# B&R Automation Studio project vibratorControlWithCurrentController (part 6)

#### Main.st - Init, cyclic, exit code
```iecst
PROGRAM _INIT

	cm.setup.name := 'sampling';

END_PROGRAM

PROGRAM _CYCLIC

	interface ACCESS ADR(gCapconInterface);

	IF gMainInterface.status.simulation OR gSimulation.status.simulateAllButWing THEN
		executeSim;
	END_IF

	IF interface.status.reset THEN
		interface.status.reset := FALSE;
		this.sim.state := 0;
	END_IF

	// ************************************************ //
	// *************** Wing Sampling ****************** //
	// ************************************************ //
	IF NOT this.hw.di_upperFlap_change THEN
		this.WingHwTOFs[0].OUT := FALSE;
	END_IF

	IF NOT this.hw.di_middleFlap_change THEN
		this.WingHwTOFs[1].OUT := FALSE;
	END_IF

	IF NOT this.hw.di_bottomFlap_change THEN
		this.WingHwTOFs[2].OUT := FALSE;
	END_IF

	IF NOT this.hw.di_neigbourFlap_change THEN
		this.WingHwTOFs[3].OUT := FALSE;
	END_IF

	FOR i:=0 TO 3 BY 1 DO
		IF NOT this.WingHwTOFs[i].OUT THEN
			this.WingHwTOFs[i].ET := this.WingHwTOFs[i].ET +1600; // 0.8 ms
		END_IF
		IF (this.WingHwTOFs[i].ET >= this.WingHwTOFs[i].PT) THEN
			CASE i OF

				0:
					IF this.hw.di_upperFlap_change THEN // only reset if changeOver signal is 1 again.
						this.WingHwTOFs[i].OUT := TRUE;
						this.WingHwTOFs[i].ET := 0;
					END_IF

				1:
					IF this.hw.di_middleFlap_change THEN // only reset if changeOver signal is 1 again.
						this.WingHwTOFs[i].OUT := TRUE;
						this.WingHwTOFs[i].ET := 0;
					END_IF

				2:
					IF this.hw.di_bottomFlap_change THEN // only reset if changeOver signal is 1 again.
						this.WingHwTOFs[i].OUT := TRUE;
						this.WingHwTOFs[i].ET := 0;
					END_IF

				3:
					IF this.hw.di_neigbourFlap_change THEN // only reset if changeOver signal is 1 again.
						this.WingHwTOFs[i].OUT := TRUE;
						this.WingHwTOFs[i].ET := 0;
					END_IF

			END_CASE
		END_IF
	END_FOR

	// ************************************************ //
	// ************** CAPCON ALGORITHM **************** //
	// ************************************************ //
	this.hw.ai_signal[0] := (this.hw.ai_signal[1]+this.lastAiSignal)/2;
	this.lastAiSignal := this.hw.ai_signal[1];
	FOR k:=0 TO 1 DO
		this.MTBasicsTimeDelay_capcon.Enable 	 := TRUE;
		this.MTBasicsTimeDelay_capcon.DelayTime  := 0.032;
		this.MTBasicsTimeDelay_capcon.In 		 := this.hw.ai_signal[k];
		this.MTBasicsTimeDelay_capcon();

		this.MTFilterMovingAverage_capcon.Enable		:= TRUE;
		this.MTFilterMovingAverage_capcon.WindowLength  := 40;
		this.MTFilterMovingAverage_capcon.In 			:= this.hw.ai_signal[k];
		this.MTFilterMovingAverage_capcon();

		this.BrickDetector_0.enable 	:= TRUE;
		this.BrickDetector_0.signal 	:= this.MTFilterMovingAverage_capcon.Out;
		this.BrickDetector_0.threshold 	:= gCapconInterface.status.capconMinThreshold;		 //15;
		this.BrickDetector_0.factorRmsMax := gCapconInterface.status.factorRmsMax;
		this.BrickDetector_0();

		this.CapconNoiseMeassure_0.beltSpeed := gBeltInterface.status.speed;
		this.CapconNoiseMeassure_0.rms := this.BrickDetector_0.rms;
		this.CapconNoiseMeassure_0();

		CASE cm.substate OF
			0:
				cm.description := 'wait for brick';

				this.BrickIntegral_0.enable := FALSE;
				this.BrickIntegral_0.calculate := FALSE;
				this.BrickIntegral_0();

				IF this.BrickDetector_0.brickCandidate AND NOT gMainInterface.status.emptying THEN
					this.BrickIntegral_0.baselineStart := this.BrickDetector_0.signal;
					cm.substate := 10;
				END_IF
			10:
				cm.description := 'measure brick';

				this.BrickIntegral_0.enable := TRUE;
				this.BrickIntegral_0.calculate := FALSE;
				this.BrickIntegral_0.signal := this.MTBasicsTimeDelay_capcon.Out;
				this.BrickIntegral_0();

				IF NOT this.BrickDetector_0.brickCandidate THEN
					cm.substate := 0;
				ELSIF this.BrickDetector_0.brickPresent THEN
					cm.substate := 20;
				END_IF

			20:
				cm.description := 'measure brick and wait for brick not present';

				this.BrickIntegral_0.enable := TRUE;
				this.BrickIntegral_0.calculate := FALSE;
				this.BrickIntegral_0.signal := this.MTBasicsTimeDelay_capcon.Out;
				this.BrickIntegral_0();

				IF this.BrickDetector_0.brickNotPresent THEN
					this.BrickIntegral_0.baselineEnd := this.BrickDetector_0.signal;
					this.BrickDetector_0.rmsMaxThreshold := this.BrickDetector_0.currentRmsMax;
					cm.substate := 30;
				END_IF

			30:
				cm.description := 'calculate integral';

				this.BrickIntegral_0.calculate := TRUE;
				this.BrickIntegral_0();

				IF this.BrickIntegral_0.done THEN
					this.BrickIntegral_0.calculate := FALSE;
					this.integralSum := this.integralSum + this.BrickIntegral_0.integral;

					cm.substate := 40;
				END_IF

			40:
				cm.description := 'Add peak integrals to array';

				IF this.BrickIntegral_0.noPeaks > 0 THEN
					FOR i:=0 TO this.BrickIntegral_0.noPeaks - 1 DO
						IF this.noPeaks <= MAX_PEAKS THEN
							this.peakIntegral[this.noPeaks] := this.BrickIntegral_0.integrals[i];
							this.noPeaks := this.noPeaks + 1;
						END_IF;
					END_FOR
				END_IF

				interface.status.noPeaks 	   := this.noPeaks;
				interface.status.peakIntegral  := this.peakIntegral;

				cm.substate := 50;

			50:
				cm.description := 'Verify peak integrals';

				this.VerifyPeaks_0.teachIntegral 	:= interface.status.teachIntegral;
				this.VerifyPeaks_0.controlPercent 	:= interface.parameter.controlPercent;
				this.VerifyPeaks_0.peakIntegral 	:= ADR(this.peakIntegral);
				this.VerifyPeaks_0.noPeaks			:= this.noPeaks;
				this.VerifyPeaks_0();

				interface.status.noVerifiedPeaks 	:= this.VerifyPeaks_0.noVerifiedPeaks;
				interface.status.verifiedPeakCount 	:= this.VerifyPeaks_0.peakCount;

				cm.substate := 60;

			60:
				cm.description := 'Verify adaptive peak integrals';

				this.VerifyPeaks_1.teachIntegral 	:= interface.status.adaptiveTeachIntegral;
				this.VerifyPeaks_1.controlPercent 	:= interface.parameter.controlPercent;
				this.VerifyPeaks_1.peakIntegral 	:= ADR(this.peakIntegral);
				this.VerifyPeaks_1.noPeaks			:= this.noPeaks;
				this.VerifyPeaks_1();

				interface.status.noAdaptiveVerifiedPeaks := this.VerifyPeaks_1.noVerifiedPeaks;

				cm.substate := 0;

		END_CASE
	END_FOR

	IF EDGEPOS(interface.status.ready) THEN
		this.integralSum := 0;
		this.brickError := FALSE;
		this.noPeaks := 0;
		this.noVerifiedPeaks := 0;
		interface.status.noPeaks := 0;
		interface.status.noVerifiedPeaks := 0;
		interface.status.noAdaptiveVerifiedPeaks := 0;
		FOR i:=0 TO MAX_PEAKS DO
			this.peakIntegral[i] := 0;
		END_FOR
	END_IF

	interface.status.integralSum := this.integralSum;
	interface.status.brickDetected := cm.substate >= 10;
	interface.status.brickPresent := cm.substate >= 20;

	// Test from FAT
	IF gCapconInterface.cmd.startSpeedSignalTest THEN
		IF NOT this.TON_0.IN THEN
			this.maxSignal := -30000;
			this.minSignal := 30000;
		END_IF

		// Save highest speed doing 5sec
		this.TON_0.PT := T#5s;
		this.TON_0.IN := TRUE;
		this.TON_0();
		this.maxSignal := SEL(this.hw.ai_signal[0]>this.maxSignal,this.maxSignal,this.hw.ai_signal[0]);
		this.minSignal := SEL(this.hw.ai_signal[0]<this.minSignal,this.minSignal,this.hw.ai_signal[0]);

		IF this.TON_0.Q THEN
			this.TON_0(IN:=FALSE);
			gCapconInterface.status.maxRawSignal := this.maxSignal-this.minSignal; // max signal peak-to-peak
			IF gCapconInterface.status.maxRawSignal > 5000 THEN
				gCapconInterface.status.maxRawSignal := 0;
			END_IF
			gCapconInterface.cmd.startSpeedSignalTest := FALSE;
		END_IF
	END_IF

END_PROGRAM

PROGRAM _EXIT

END_PROGRAM
```

#### executeSim.st
```iecst
ACTION executeSim:

	this.hw.ai_signal[1] := gSimCapcon.status.simSignal;

END_ACTION
```

#### Types.typ - Local data types
```iecst
TYPE
	local_alarm_typ : 	STRUCT
		noisePeakPeak : BOOL;
		noiseOffset : BOOL;
		noiseSpeed : BOOL;
	END_STRUCT;
	local_TOF_typ : 	STRUCT
		PT : UDINT := 10000; (*10ms*)
		ET : UDINT;
		OUT : BOOL;
	END_STRUCT;
	local_brickDetect_typ : 	STRUCT
		state : USINT;
		stateDescription : STRING[200];
	END_STRUCT;
	local_typ : 	STRUCT
		hw : local_hw_typ;
		sim : local_sim_typ;
		WingHwTOFs : ARRAY[0..3]OF local_TOF_typ;
		TON_timeout : TON;
		alarm : local_alarm_typ;
		BrickDetector_0 : BrickDetector;
		BrickIntegral_0 : BrickIntegral;
		integralSum : REAL;
		peakIntegral : ARRAY[0..MAX_PEAKS]OF REAL;
		noPeaks : USINT;
		noVerifiedPeaks : USINT;
		brickError : BOOL := FALSE;
		tmpBrickCount : USINT;
		MTBasicsTimeDelay_capcon : MTBasicsTimeDelay;
		MTFilterMovingAverage_capcon : MTFilterMovingAverage;
		upperIntegralLimit : REAL;
		lowerIntegralLimit : REAL;
		VerifyPeaks_1 : VerifyPeaks;
		VerifyPeaks_0 : VerifyPeaks;
		TON_capconNoise : TON;
		MTDataMinMax_0 : MTDataMinMax;
		CapconNoiseMeassure_0 : CapconNoiseMeassure;
		lastAiSignal : INT;
		TON_0 : TON;
		maxSignal : REAL;
		minSignal : REAL;
	END_STRUCT;
	local_hw_typ : 	STRUCT
		ai_signal : ARRAY[0..1]OF INT; (*Signal name: AI_CCH
PJ95: B400
Connector: AI.01
Description: Analogue signal from Capcon head.*)
		di_middleFlap_change : BOOL;
		di_neigbourFlap_change : BOOL;
		di_bottomFlap_change : BOOL;
		di_upperFlap_change : BOOL;
	END_STRUCT;
	local_sim_typ : 	STRUCT
		state : UDINT;
		sampleCount : DINT;
		recordCount : DINT;
		sampleDelay : local_time_typ;
	END_STRUCT;
	local_taskTime_typ : 	STRUCT
		time : UDINT;
		elapsed : UDINT;
		maximum : UDINT;
	END_STRUCT;
END_TYPE
```

#### Variables.var - Local variables
```iecst
VAR
	cm : brdkCM;
	i : USINT;
	interface : REFERENCE TO gCapconInterface_typ;
	this : local_typ;
	k : USINT;
END_VAR
```

#### LocalFunctions.fun
```iecst
FUNCTION_BLOCK VerifyPeaks
	VAR_INPUT
		teachIntegral : REAL;
		controlPercent : USINT;
		peakIntegral : REFERENCE TO ARRAY[0..MAX_PEAKS] OF REAL;
		noPeaks : UINT;
	END_VAR
	VAR_OUTPUT
		noVerifiedPeaks : USINT;
		peakCount : ARRAY[0..MAX_PEAKS] OF USINT;
	END_VAR
	VAR
		j : UINT;
		i : UINT;
		upperIntegralLimit : REAL;
		lowerIntegralLimit : REAL;
	END_VAR
END_FUNCTION_BLOCK

FUNCTION_BLOCK BrickDetector
	VAR_INPUT
		enable : BOOL;
		signal : REAL;
		threshold : REAL; (*Rms threshold for when it is considered a brick*)
		factorRmsMax : REAL := 0.001;
		rmsMaxThreshold : REAL;
	END_VAR
	VAR_OUTPUT
		ready : BOOL;
		rms : REAL;
		slope : REAL;
		brickPresent : BOOL;
		brickNotPresent : BOOL;
		brickCandidate : BOOL;
		currentRmsMax : REAL;
	END_VAR
	VAR
		rmsThreshold : REAL;
		fifoIdx : UDINT;
		endIdx : UDINT;
		buffer : ARRAY[0..49] OF REAL;
		a : REAL;
		b : REAL;
		i : UDINT;
		rmsMax : REAL;
		presentCounter : UDINT;
	END_VAR
END_FUNCTION_BLOCK

FUNCTION_BLOCK BrickIntegral
	VAR_INPUT
		enable : BOOL; (*Enable function block and start buffering signal*)
		calculate : BOOL; (*Integral calculated when true*)
		signal : REAL;
		baselineStart : REAL;
		baselineEnd : REAL;
	END_VAR
	VAR_OUTPUT
		done : BOOL;
		integral : REAL; (*The integral calculated when calculate is true*)
		bufferSize : UINT;
		bufferFull : BOOL; (*The internal buffer is full and the integral is wrong after this point*)
		noPeaks : USINT;
		peakIntegrals : ARRAY[0..MAX_PEAKS] OF REAL;
		integrals : ARRAY[0..MAX_PEAKS] OF REAL;
		startDive : REAL;
		highestPeak : REAL;
	END_VAR
	VAR
		state : UINT;
		buffer : ARRAY[0..2500] OF REAL;
		bufferIdx : UINT;
		currBufferIdx : UINT;
		i : UINT;
		j : UINT;
		a : REAL;
		b : REAL;
		totalPeakIntegral : REAL;
		peakStart : ARRAY[0..MAX_PEAKS] OF UINT;
		peakEnd : ARRAY[0..MAX_PEAKS] OF UINT;
		startDives : ARRAY[0..MAX_PEAKS] OF REAL;
		startIdx : UINT;
		endIdx : UINT;
		sortedNoPeaks : USINT;
		oldEnable : BOOL;
		firstDive : BOOL;
		lastHighestPeak : REAL;
	END_VAR
END_FUNCTION_BLOCK

FUNCTION_BLOCK CapconNoiseMeassure
	VAR_INPUT
		beltSpeed : LEGO_SPEED_ENUM;
		rms : REAL;
	END_VAR
	VAR_OUTPUT
		Out : REAL;
	END_VAR
	VAR
		MTDataMinMax_0 : MTDataMinMax;
		state : USINT;
		TON_0 : TON;
	END_VAR
END_FUNCTION_BLOCK
```

#### LocalFunctions.st
```iecst
(* TODO: Add your comment here *)
FUNCTION_BLOCK BrickDetector
	brickPresent := FALSE;
	brickNotPresent := FALSE;
	IF enable THEN
		buffer[fifoIdx] := signal;
		endIdx := fifoIdx;
		IF fifoIdx = RMS_BUFFER_LEN THEN
			fifoIdx := 0;
			ready := TRUE;
		ELSE
			fifoIdx := fifoIdx + 1;
		END_IF
		IF ready THEN
			a := (buffer[endIdx]-buffer[fifoIdx])/ USINT_TO_REAL(RMS_BUFFER_LEN);
			b := buffer[fifoIdx];
			rms := 0;
			FOR i:=0 TO RMS_BUFFER_LEN DO
				rms := rms + EXPT((buffer[(fifoIdx+i) MOD (RMS_BUFFER_LEN+1)]) - (a*UDINT_TO_REAL(i)+b), 2);
			END_FOR
			rms := rms / USINT_TO_REAL(RMS_BUFFER_LEN + 1);

			IF rms > rmsMax THEN
				rmsMax := rms;
			END_IF

			slope := a;
			rmsThreshold := LIMIT(threshold,rmsMaxThreshold*factorRmsMax,450);

			IF rms < rmsThreshold AND ABS(slope) < 1 THEN
				brickCandidate := FALSE;
			END_IF

			IF rms > rmsThreshold THEN
				brickCandidate := TRUE;
				presentCounter := SEL(presentCounter >= RMS_COUNT_THRESHOLD, presentCounter + 1, RMS_COUNT_THRESHOLD);
				IF presentCounter >= RMS_COUNT_THRESHOLD AND rmsMax > 500 THEN
					brickPresent := TRUE;
				ELSIF presentCounter > 250 THEN
					brickCandidate := FALSE;
					presentCounter := 0;
				END_IF
			ELSIF rms < rmsThreshold AND ABS(slope) < 2.5 THEN
				presentCounter := SEL(presentCounter = 0, presentCounter - 1, 0);
				IF presentCounter = 0 THEN
					brickNotPresent := TRUE;
					brickCandidate := FALSE;
					currentRmsMax := rmsMax;
					rmsMax := 0;
				END_IF
			END_IF
		END_IF
	ELSE
		fifoIdx := 0;
		ready := FALSE;
		brickCandidate := FALSE;
	END_IF
END_FUNCTION_BLOCK

FUNCTION_BLOCK BrickIntegral
	IF enable THEN
		IF NOT bufferFull THEN
			buffer[bufferIdx] := signal;
			IF bufferIdx < 1250 THEN
				bufferIdx := bufferIdx + 1;
			ELSE
				bufferFull := TRUE;
			END_IF
		END_IF

		CASE state OF
			0:
				IF calculate THEN
					IF bufferIdx > RMS_COUNT_THRESHOLD+1 THEN
						a := (baselineEnd-baselineStart)/(bufferIdx-RMS_COUNT_THRESHOLD+1);
						b := baselineStart;
						startDive := buffer[0];
						firstDive := TRUE;
						highestPeak := buffer[0];
						currBufferIdx := 0;
						state := 10;
					ELSE
						state := 100;
					END_IF
				END_IF

			10:
				FOR i:=currBufferIdx TO bufferIdx-RMS_COUNT_THRESHOLD+1 DO
					IF (a*i+b) - buffer[i] > startDive AND firstDive THEN
						startDive := (a*i+b) - buffer[i];
					END_IF
					IF buffer[i] > highestPeak THEN
						highestPeak := buffer[i];
					END_IF
					IF buffer[i] - baselineStart > lastHighestPeak * 0.2 THEN
						firstDive := FALSE;
					END_IF
					IF buffer[i] > (a*i+b) THEN
						peakIntegrals[noPeaks] := peakIntegrals[noPeaks] + buffer[i] - (a*i+b);
						IF peakStart[noPeaks] = 0 THEN
							peakStart[noPeaks] := i;
						END_IF
					ELSE
						IF peakIntegrals[noPeaks] < 500 THEN
							peakIntegrals[noPeaks] := 0;
						ELSE
							peakEnd[noPeaks] := i;
							startDives[noPeaks] := startDive;
							totalPeakIntegral := peakIntegrals[noPeaks];
							noPeaks := MIN(noPeaks + 1, MAX_PEAKS);
							firstDive := TRUE;
							startDive := 0;
						END_IF
					END_IF

					integral := integral + buffer[i] - (a*i+b-startDive);

					IF i >= currBufferIdx + 100 THEN
						currBufferIdx := i;
						EXIT;
					END_IF
				END_FOR

				IF i > bufferIdx-RMS_COUNT_THRESHOLD+1 THEN
					state := 20;
				END_IF

			20:
				// Remove small integrals
				sortedNoPeaks := 0;
				IF noPeaks > 0 AND totalPeakIntegral <> 0 THEN
					FOR j:=0 TO noPeaks-1 DO
						IF peakIntegrals[j] / totalPeakIntegral > 0.05 THEN
							peakIntegrals[sortedNoPeaks] := peakIntegrals[j];
							peakStart[sortedNoPeaks] := peakStart[j];
							peakEnd[sortedNoPeaks] := peakEnd[j];
							startDives[sortedNoPeaks] := startDives[j];
							sortedNoPeaks := sortedNoPeaks + 1;
						END_IF
					END_FOR
				END_IF

				state := 30;

			30:
				// Calculate integral for each peak
				IF sortedNoPeaks > 0 THEN
					FOR j:=0 TO sortedNoPeaks-1 DO
						// Find start index
						IF j = 0 THEN
							startIdx := peakStart[j];
						ELSE
							startIdx := peakStart[j] - (peakStart[j]-peakEnd[j-1])/2;
						END_IF
						// Find end index
						IF j = sortedNoPeaks-1 THEN
							endIdx := peakEnd[j];
						ELSE
							endIdx := peakEnd[j] + (peakStart[j+1]-peakEnd[j])/2;
						END_IF
						startDive := startDives[j];
						FOR i:=startIdx TO endIdx DO
							integrals[j] := integrals[j] + buffer[i] - (a*i+b-startDive);
						END_FOR
					END_FOR
				END_IF

				noPeaks := sortedNoPeaks;

				state := 100;

			100:
				done := TRUE;

				IF NOT calculate THEN
					done := FALSE;
					lastHighestPeak := highestPeak;
					state := 0;
				END_IF

		END_CASE
		oldEnable := TRUE;
	ELSIF oldEnable THEN
		bufferIdx := 0;
		integral := 0;
		noPeaks := 0;
		sortedNoPeaks := 0;
		totalPeakIntegral := 0;
		FOR i:=0 TO MAX_PEAKS DO
			peakIntegrals[i] := 0;
			integrals[i] := 0;
			peakStart[i] := 0;
			peakEnd[i] := 0;
			startDives[i] := 0;
		END_FOR

		bufferFull := FALSE;
		oldEnable := FALSE;
	END_IF
	bufferSize := bufferIdx;
END_FUNCTION_BLOCK

FUNCTION_BLOCK VerifyPeaks

	noVerifiedPeaks := 0;
	brsmemset(ADR(peakCount), 0, SIZEOF(peakCount));
	IF noPeaks > 0 THEN
		FOR i:=0 TO noPeaks-1 DO
			FOR j:=1 TO 6 DO
				IF j > 1 AND controlPercent < 50 THEN
					lowerIntegralLimit := upperIntegralLimit;
				ELSE
					lowerIntegralLimit := (teachIntegral*UINT_TO_REAL(j))-(teachIntegral*(USINT_TO_REAL((controlPercent))/100.0));
				END_IF
				upperIntegralLimit := (teachIntegral*UINT_TO_REAL(j))+(teachIntegral*(USINT_TO_REAL(controlPercent)/100.0));
				IF peakIntegral[i] > lowerIntegralLimit AND peakIntegral[i] <= upperIntegralLimit THEN
					noVerifiedPeaks := noVerifiedPeaks + DINT_TO_USINT(j);
					peakCount[i] := DINT_TO_USINT(j);
					EXIT;
				END_IF
			END_FOR
			IF peakIntegral[i] >= (teachIntegral*6)+(teachIntegral*(USINT_TO_REAL(controlPercent)/100.0)) THEN
				noVerifiedPeaks := noVerifiedPeaks + 7;
				peakCount[i] := 7;
			END_IF
		END_FOR
	END_IF

END_FUNCTION_BLOCK

FUNCTION_BLOCK CapconNoiseMeassure

	CASE state OF

		0:
			TON_0.IN := beltSpeed = lego_speed_stop;
			TON_0.PT := T#10s;
			TON_0();

			IF TON_0.Q THEN
				TON_0.IN := FALSE;
				TON_0();
				MTDataMinMax_0.Enable := FALSE;
				MTDataMinMax_0();
				state := 10;
			END_IF

		10:

			MTDataMinMax_0.Enable := TRUE;
			MTDataMinMax_0.In := rms;
			MTDataMinMax_0();

			TON_0.IN := TRUE;
			TON_0.PT := T#1s;
			TON_0();

			IF beltSpeed <> lego_speed_stop THEN
				TON_0.IN := FALSE;
				TON_0();
				state := 0;
			ELSIF TON_0.Q THEN
				TON_0.IN := FALSE;
				TON_0();

				Out := MTDataMinMax_0.MaxValue;
				state := 0;
			END_IF

	END_CASE

END_FUNCTION_BLOCK
```

#### LocalFunctions.var
```iecst
VAR CONSTANT
	RMS_BUFFER_LEN : USINT := 40;
	RMS_COUNT_THRESHOLD : USINT := 10;
END_VAR
```

### Program Logical/modules/feeder/feeder (IEC)

#### producing.st
```iecst
ACTION producing:

	CASE em.state OF

		STATE_STOPPED:

			em.description := 'Waiting for start command';
			em.cmd.reset 	:= interface.cmd.start OR this.hmi.cmd.empty;
			IF gConfig.status.loadInitialValue[0] AND (gRecipe.status.saved OR gRecipe.status.loaded) AND (gConfig.status.saved OR gConfig.status.loaded) THEN
				gConfig.status.loadInitialValue[0] := FALSE;
				recipe.offTime := 1000;
				recipe.onTime := 1000;
				recipe.startDelay := 30;
				recipe.stopDelay := 30;
			END_IF
			IF this.hmi.cmd.forceForwards AND this.hmi.cmd.forceBackwards THEN
				this.hmi.cmd.forceForwards := FALSE;
				this.hmi.cmd.forceBackwards := FALSE;
			END_IF
			this.belt.cmd.forwards := this.hmi.cmd.forceForwards;
			this.belt.cmd.backwards := this.hmi.cmd.forceBackwards;

			em.cmd.sc 		:= TRUE;

		STATE_IDLE:

			em.cmd.start := em.cmd.sc := TRUE;

		STATE_STARTING:

			em.description := 'wait for feeder flap to close';
			IF this.flap.state = FEEDER_FLAP_CLOSED THEN
				this.flap.cmd.close := FALSE;
				this.stopCounter := 0;
				this.startCounter := 0;
				this.onCounter := 0;
				this.offCounter := 0;
				em.cmd.sc := TRUE;
			ELSE
				this.flap.cmd.close := TRUE;
			END_IF

		STATE_EXECUTE:

			this.hmi.status.running := interface.status.running := this.hmi.cmd.enable;		// running if enabled from HMI

			IF this.flap.state <> FEEDER_FLAP_CLOSED OR gFeederInterface.cmd.stop OR this.hmi.cmd.stop THEN
				this.hmi.cmd.stop := FALSE;
				em.cmd.stop := TRUE;
			END_IF

			CASE em.substate OF
				0:
					em.description := 'wait for CF running and low level';

					IF cmIsRunning(interface.cmd.speed) AND NOT this.hw.di_levelSensorInBowl THEN
						em.substate := 10;
					END_IF

				10:
					em.description := 'wait start delay';

					this.startCounter := this.startCounter + 1;

					IF this.hw.di_levelSensorInBowl THEN
						this.startCounter := 0;
						em.substate := 0;
					ELSIF NOT cmIsRunning(interface.cmd.speed) THEN
						em.substate := 0;
					ELSIF UDINT_TO_REAL(this.startCounter*this.RTInfo_0.cycle_time)/1000.0 > recipe.startDelay THEN
						this.belt.cmd.forwards := TRUE;
						this.startCounter := 0;
						em.substate := 20;
					END_IF

				20:
					em.description := 'belt running for on time';

					this.onCounter := this.onCounter + 1;

					IF this.hw.di_levelSensorInBowl THEN
						this.belt.cmd.forwards := FALSE;
						em.substate := 40;
					ELSIF NOT cmIsRunning(interface.cmd.speed) THEN
						this.onCounter := 0;
						this.belt.cmd.forwards := FALSE;
						em.substate := 0;
					ELSIF UDINT_TO_REAL(this.onCounter*this.RTInfo_0.cycle_time)/1000.0 > recipe.onTime THEN
						this.onCounter := 0;
						this.belt.cmd.forwards := FALSE;
						em.substate := 30;
					END_IF

				30:
					em.description := 'belt stopped for off time';

					this.offCounter := this.offCounter + 1;

					IF NOT cmIsRunning(interface.cmd.speed) THEN
						this.offCounter := 0;
						em.substate := 0;
					ELSIF UDINT_TO_REAL(this.offCounter*this.RTInfo_0.cycle_time)/1000.0 > recipe.offTime THEN
						this.offCounter := 0;

						this.belt.cmd.forwards := TRUE;
						em.substate := 20;
					END_IF

				40:
					em.description := 'wait for stop delay';

					this.stopCounter := this.stopCounter + 1;

					IF UDINT_TO_REAL(this.stopCounter*this.RTInfo_0.cycle_time)/1000.0 > recipe.stopDelay OR NOT cmIsRunning(interface.cmd.speed) THEN
						this.stopCounter := 0;
						em.substate := 0;
					ELSIF NOT this.hw.di_levelSensorInBowl THEN
						this.stopCounter := 0;
						this.belt.cmd.forwards := TRUE;
						em.substate := 20;
					END_IF

			END_CASE

			em.cmd.complete := this.hmi.cmd.empty;
			em.cmd.sc := TRUE;

		STATE_SUSPENDED:

			em.cmd.sc := TRUE;

		STATE_COMPLETING:

			this.hmi.cmd.empty := FALSE;

			CASE em.substate OF

				0:
					em.description := 'waiting for an empty box at the flap';

					this.belt.cmd.backwards := this.belt.cmd.forwards := this.flap.cmd.open := this.flap.cmd.close := FALSE;

					IF this.hw.di_boxIsReadyAtFlap THEN
						this.alarm.boxMissing.active := FALSE;
						em.substate := 10;
					ELSE
						IF NOT this.hmi.cmd.confirmEmpty THEN
							this.alarm.boxMissing.active := TRUE;
						ELSE	// If user confirm -> exit COMPLETING and be ready for production.
							this.alarm.boxMissing.active := FALSE;
							em.cmd.sc := TRUE;
						END_IF
					END_IF

				10:
					em.description := 'flap opening';

					this.flap.cmd.open := TRUE;

					IF this.flap.state = FEEDER_FLAP_OPENED THEN
						this.flap.cmd.open := FALSE;
						this.TON_startDelay(IN :=FALSE);
						this.TON_startDelay.PT := T#2s;
						em.substate := 20;
					END_IF

				20:
					em.description := 'run belt backwards until box is removed';

					// Run the belt backwards 10s then stop 2s etc. etc. This is done not to burn card.
					this.TON_startDelay.IN := TRUE;
					this.TON_startDelay();
					IF this.TON_startDelay.Q THEN
						this.TON_startDelay(IN:=FALSE);
						IF this.belt.cmd.backwards THEN
							// if it has just been running wait 2s
							this.TON_startDelay.PT := T#2s;
						ELSE
							// If it has not been running - run it for 10s
							this.TON_startDelay.PT := T#10s;
						END_IF
						this.belt.cmd.backwards := NOT this.belt.cmd.backwards;
					END_IF

					IF NOT this.hw.di_boxIsReadyAtFlap THEN
						this.belt.cmd.backwards := FALSE;
						this.TON_startDelay(IN :=FALSE);
						em.substate := 25;
					END_IF

				25:
					em.description := 'Wait 3s before moving from backward to forward to avoid huge current peak';
					this.TON_startDelay.IN := TRUE;
					this.TON_startDelay.PT := T#3s;
					this.TON_startDelay();

					IF this.TON_startDelay.Q THEN
						this.TON_startDelay(IN:=FALSE);
						em.substate := 30;
					END_IF

				30:
					em.description := 'flap closing and run belt forward';

					this.belt.cmd.forwards := this.flap.cmd.close := TRUE;

					IF this.flap.state = FEEDER_FLAP_CLOSED THEN
						this.flap.cmd.close := this.belt.cmd.forwards :=  FALSE;
						em.cmd.sc := TRUE;
					END_IF

			END_CASE

		STATE_COMPLETE:

			this.belt.cmd.backwards := this.belt.cmd.forwards := this.flap.cmd.open := this.flap.cmd.close := this.hmi.cmd.confirmEmpty := FALSE;
			em.cmd.stop := em.cmd.sc := TRUE;

		STATE_STOPPING, STATE_HOLDING, STATE_ABORTING, STATE_RESETTING, STATE_SUSPENDING:

			em.description := 'close flap with max speed and check belt type';

			this.belt.cmd.backwards := this.belt.cmd.forwards := this.flap.cmd.open := this.flap.cmd.close := this.hmi.cmd.confirmEmpty := this.hmi.cmd.forceForwards := this.hmi.cmd.forceBackwards := FALSE;

			interface.status.count := 0;
			this.hmi.status.running	:= interface.status.running := FALSE;
			this.TON_timeout(IN := FALSE);
			this.TON_startDelay(IN := FALSE);
			this.flap.cmd.open := FALSE;
			em.cmd.sc := TRUE;

		STATE_ABORTED:

			IF NOT MpAlarmXCheckReaction(mpAlarmXCore,'abortFeeder') THEN
				em.cmd.clear := em.cmd.sc := TRUE;
			END_IF

		STATE_CLEARING:

			CASE em.substate OF

				0:
					brsmemset(ADR(this.alarm), 0, SIZEOF(this.alarm));
					// Set alarm texts
					this.alarm.lowLevel.name := 'feederLowLevel';
					this.alarm.boxMissing.name := 'feederBoxMissing';
					this.alarm.cannotCloseFlap.name := 'feederCannotCloseFlap';
					this.alarm.cannotOpenFlap.name := 'feederCannotOpenFlap';
					this.alarm.beltFeederEmpty.name := 'beltFeederEmpty';
					em.substate := 10;

				10:
					this.TON_timeout(IN := TRUE);
					IF this.flap.state = FEEDER_FLAP_CLOSED OR  this.TON_timeout.Q THEN
						this.TON_timeout(IN := FALSE);
						this.flap.cmd.close := FALSE;

						em.cmd.sc := TRUE;
					ELSE
						this.flap.cmd.close := TRUE;
					END_IF

			END_CASE

		ELSE

			em.cmd.sc := TRUE;

	END_CASE

	END_ACTION
```

#### flapAndBeltControl.st
```iecst
ACTION flapControl:

	this.flap.internal.TON_delaySwitch.PT  := T#100ms;
	this.flap.internal.TON_maxOpenTime.PT  := config.maxOpenCloseTime;
	this.flap.internal.TON_maxCloseTime.PT := config.maxOpenCloseTime;
	this.flap.internal.TON_overCurrentProtect.PT := config.overCurrentProtectTime;

	IF this.flap.state <> this.flap.internal.oldState THEN

		this.flap.internal.TON_delaySwitch(IN:=FALSE);
		this.flap.internal.TON_maxOpenTime(IN:=FALSE);
		this.flap.internal.TON_maxCloseTime(IN:=FALSE);
		this.flap.internal.TON_overCurrentProtect(IN:=FALSE);
		this.flap.internal.oldState := this.flap.state;
	END_IF

	flapOpening := this.hw.do_flapOpen;
	flapClosing := this.hw.do_flapClose;

	CASE this.flap.state OF

		FEEDER_FLAP_IDLE:

			this.hw.do_flapOpen := this.hw.do_flapClose := FALSE;

			IF this.flap.cmd.open THEN
				this.flap.state := FEEDER_FLAP_OPENING;
			ELSIF this.flap.cmd.close THEN
				this.flap.state := FEEDER_FLAP_CLOSING;
			ELSE
				IF NOT this.hw.di_flapIsOpen THEN
					this.flap.state := FEEDER_FLAP_OPENED;
				ELSIF this.hw.di_flapIsClosed THEN
					this.flap.state := FEEDER_FLAP_CLOSED;
				END_IF
			END_IF

		FEEDER_FLAP_OPENING:

			this.hw.do_flapClose := this.flap.cmd.close := FALSE;

			IF NOT this.hw.di_flapIsOpen THEN
				this.hw.do_flapOpen := this.flap.cmd.open := FALSE;
				this.flap.state := FEEDER_FLAP_OPENED;
			ELSIF this.flap.cmd.open THEN
				this.flap.internal.TON_maxOpenTime(IN := TRUE);
				this.hw.do_flapOpen := TRUE;
				this.flap.internal.TON_overCurrentProtect(IN := this.hw.di_flapIsClosed);
			ELSE
				this.flap.internal.TON_delaySwitch(IN := TRUE);
				this.hw.do_flapOpen := FALSE;
				IF this.flap.internal.TON_delaySwitch.Q THEN
					this.flap.internal.TON_delaySwitch(IN := FALSE);
					this.flap.internal.TON_maxOpenTime(IN := FALSE);
					this.flap.internal.TON_overCurrentProtect(IN := FALSE);
					this.flap.state := FEEDER_FLAP_IDLE;
				END_IF
			END_IF

			IF this.flap.internal.TON_maxOpenTime.Q OR this.flap.internal.TON_overCurrentProtect.Q THEN
				this.flap.internal.TON_maxOpenTime(IN := FALSE);
				this.flap.internal.TON_overCurrentProtect(IN := FALSE);
				this.hw.do_flapOpen := FALSE;
				this.alarm.cannotOpenFlap.active := TRUE;
				this.flap.state := FEEDER_FLAP_IDLE;
			END_IF

		FEEDER_FLAP_OPENED:

			this.hw.do_flapOpen := FALSE;

			IF this.hw.di_flapIsOpen THEN
				this.flap.state := FEEDER_FLAP_IDLE;
			ELSIF this.flap.cmd.close AND NOT this.flap.cmd.open THEN
				this.flap.state := FEEDER_FLAP_CLOSING;
			END_IF

		FEEDER_FLAP_CLOSING:

			this.hw.do_flapOpen := this.flap.cmd.open := FALSE;

			IF this.hw.di_flapIsClosed THEN
				this.hw.do_flapClose := this.flap.cmd.close := FALSE;
				this.flap.state := FEEDER_FLAP_CLOSED;
			ELSIF this.flap.cmd.close THEN
				this.flap.internal.TON_maxCloseTime(IN := TRUE);
				this.hw.do_flapClose := TRUE;
				this.flap.internal.TON_overCurrentProtect(IN := NOT this.hw.di_flapIsOpen);
			ELSE
				this.flap.internal.TON_delaySwitch(IN := TRUE);
				this.hw.do_flapClose := FALSE;
				IF this.flap.internal.TON_delaySwitch.Q THEN
					this.flap.internal.TON_delaySwitch(IN := FALSE);
					this.flap.internal.TON_maxCloseTime(IN := FALSE);
					this.flap.internal.TON_overCurrentProtect(IN := FALSE);
					this.flap.state := FEEDER_FLAP_IDLE;
				END_IF
			END_IF

			IF this.flap.internal.TON_maxCloseTime.Q OR this.flap.internal.TON_overCurrentProtect.Q THEN
				this.flap.internal.TON_maxCloseTime(IN := FALSE);
				this.flap.internal.TON_overCurrentProtect(IN := FALSE);
				this.hw.do_flapClose := FALSE;
				this.alarm.cannotCloseFlap.active := TRUE;
				this.flap.state := FEEDER_FLAP_IDLE;
			END_IF

		FEEDER_FLAP_CLOSED:

			this.hw.do_flapClose := FALSE;

			IF NOT this.hw.di_flapIsClosed THEN
				this.flap.state := FEEDER_FLAP_IDLE;
			ELSIF this.flap.cmd.open AND NOT this.flap.cmd.close THEN
				this.flap.state := FEEDER_FLAP_OPENING;
			END_IF

	END_CASE

	this.hmi.status.flapOpen := this.flap.state = FEEDER_FLAP_OPENED;
	this.hmi.status.flapClose := this.flap.state = FEEDER_FLAP_CLOSED;

END_ACTION

ACTION beltControl:

	this.belt.internal.TON_delaySwitch.PT := T#1000ms;

	CASE this.belt.state OF

		FEEDER_BELT_IDLE:

			this.hw.do_beltBackwards := this.hw.do_beltForwards := FALSE;

			IF this.belt.cmd.forwards THEN
				this.belt.state := FEEDER_BELT_FORWARDS;
			ELSIF this.belt.cmd.backwards THEN
				this.belt.state := FEEDER_BELT_BACKWARDS;
			END_IF

		FEEDER_BELT_FORWARDS:

			this.hw.do_beltBackwards := FALSE;

			IF this.belt.cmd.forwards THEN
				this.hw.do_beltForwards := (this.hmi.cmd.enable AND gCapconInterface.status.numBricksInPortion > 0) OR this.hmi.cmd.forceForwards;			// Only run if enabled on HMI
			ELSE
				this.hw.do_beltForwards := FALSE;
				this.belt.internal.TON_delaySwitch(IN := TRUE);
				IF this.belt.internal.TON_delaySwitch.Q THEN
					this.belt.internal.TON_delaySwitch(IN := FALSE);
					this.belt.state := FEEDER_BELT_IDLE;
				END_IF
			END_IF

		FEEDER_BELT_BACKWARDS:

			this.hw.do_beltForwards := FALSE;

			IF this.belt.cmd.backwards THEN
				this.hw.do_beltBackwards := TRUE;
			ELSE
				this.hw.do_beltBackwards := FALSE;
				this.belt.internal.TON_delaySwitch(IN := TRUE);
				IF this.belt.internal.TON_delaySwitch.Q THEN
					this.belt.internal.TON_delaySwitch(IN := FALSE);
					this.belt.state := FEEDER_BELT_IDLE;
				END_IF
			END_IF

	END_CASE

	END_ACTION
```

#### alarm.st
```iecst
ACTION alarm:

	// Low level
	this.TON_lowLevel(IN := NOT this.hw.di_levelSensorBelt AND em.state <> STATE_STOPPED, PT := T#2s);
	this.alarm.lowLevel.active := this.TON_lowLevel.Q;

	IF this.alarm.lowLevel.active AND NOT this.alarm.lowLevel.oldActive THEN
		this.alarm.lowLevel.instanceID := MpAlarmXSet(mpAlarmXCore, this.alarm.lowLevel.name);
	ELSIF this.alarm.lowLevel.oldActive AND NOT this.alarm.lowLevel.active THEN
		MpAlarmXAcknowledgeID(mpAlarmXCore, this.alarm.lowLevel.instanceID);
	END_IF
	this.alarm.lowLevel.oldActive := this.alarm.lowLevel.active;

//	IF this.hw.di_levelSensorBelt THEN
//		this.alarm.lowLevel.active := FALSE;
//		this.lowLevelTime := 0;
//	ELSIF this.belt.state = FEEDER_BELT_FORWARDS THEN
//		this.lowLevelTime := this.lowLevelTime + em.status.cycleTime;
//
//		IF this.lowLevelTime >= config.alarmLowLevelTime THEN
//			this.alarm.lowLevel.active := TRUE;
//		END_IF
//	END_IF

	// Box Missing

	IF this.alarm.boxMissing.active AND NOT this.alarm.boxMissing.oldActive THEN
		this.alarm.boxMissing.instanceID := MpAlarmXSet(mpAlarmXCore, this.alarm.boxMissing.name);
	ELSIF this.alarm.boxMissing.oldActive AND NOT this.alarm.boxMissing.active THEN
		MpAlarmXAcknowledgeID(mpAlarmXCore, this.alarm.boxMissing.instanceID);
	END_IF
	this.alarm.boxMissing.oldActive := this.alarm.boxMissing.active;

	// Cannot Close Flap
	IF gAlarm.status.ready THEN
		IF this.alarm.cannotCloseFlap.active AND NOT this.alarm.cannotCloseFlap.oldActive THEN
			this.alarm.cannotCloseFlap.instanceID := MpAlarmXSet(mpAlarmXCore, this.alarm.cannotCloseFlap.name);
		END_IF
		this.alarm.cannotCloseFlap.oldActive := this.alarm.cannotCloseFlap.active;
	END_IF

	// Cannot Open Flap
	IF gAlarm.status.ready THEN
		IF this.alarm.cannotOpenFlap.active AND NOT this.alarm.cannotOpenFlap.oldActive THEN
			this.alarm.cannotOpenFlap.instanceID := MpAlarmXSet(mpAlarmXCore, this.alarm.cannotOpenFlap.name);
		END_IF
		this.alarm.cannotOpenFlap.oldActive := this.alarm.cannotOpenFlap.active AND gAlarm.status.ready;
	END_IF

	// Belt feeder empty

	IF this.alarm.beltFeederEmpty.active AND NOT this.alarm.beltFeederEmpty.oldActive THEN
		this.alarm.beltFeederEmpty.instanceID := MpAlarmXSet(mpAlarmXCore, this.alarm.cannotOpenFlap.name);
	END_IF
	this.alarm.beltFeederEmpty.oldActive := this.alarm.beltFeederEmpty.active;

	(****************************** REACTION ******************************)
	IF em.state <> STATE_ABORTED AND em.state <> STATE_ABORTING AND em.state <> STATE_CLEARING THEN
		IF MpAlarmXCheckReaction(mpAlarmXCore,'abortFeeder') THEN
			em.cmd.abort := TRUE;
		END_IF
	END_IF
	(**********************************************************************)

END_ACTION
```

#### feeder.st - Init, cyclic, exit code
```iecst
PROGRAM _INIT

	em.setup.name := 'feeder';
	em.setup.lastActivated := FALSE;

	// gets the task name and setup names for config and receipe types
	ST_name(0,ADR(this.configName),0);
	brdkStrCpy(ADR(this.recipeName),ADR(this.configName));
	brdkStrCpy(ADR(this.recipeNameCurrent),ADR(this.configName));
	brdkStrCat(ADR(this.configName),ADR(':this.hmi.config'));
	brdkStrCat(ADR(this.recipeName),ADR(':this.hmi.recipe'));
	brdkStrCat(ADR(this.recipeNameCurrent),ADR(':this.hmi.recipeCurrent'));

	setupPointers;

	this.hmi.cmd.enable := TRUE;			// always enable BF on a boot.

	// Set alarm texts
	this.alarm.lowLevel.name := 'feederLowLevel';
	this.alarm.boxMissing.name := 'feederBoxMissing';
	this.alarm.cannotCloseFlap.name := 'feederCannotCloseFlap';
	this.alarm.cannotOpenFlap.name := 'feederCannotOpenFlap';
	this.alarm.beltFeederEmpty.name := 'beltFeederEmpty';

	this.alarm.cannotCloseFlap.active := flapClosing;
	this.alarm.cannotOpenFlap.active := flapOpening;

END_PROGRAM

PROGRAM _CYCLIC

	setupPointers;

	this.hw.do_levelSensorInBowlLow 	:= recipe.levelSensor = LEVEL_SENSOR_LOW;
	this.hw.do_levelSensorInBowlMedium 	:= recipe.levelSensor = LEVEL_SENSOR_MEDIUM;
	this.hw.do_levelSensorInBowlHigh 	:= recipe.levelSensor = LEVEL_SENSOR_HIGH;

	IF interface.cmd.empty THEN // Signal from OPCUA to empty feeder
		interface.cmd.empty := FALSE;
		this.hmi.cmd.empty := TRUE;
	END_IF

	// Signal indicator for when vibrator is empty
	this.TON_VibratorBowlEmpty.IN := NOT this.hw.di_levelSensorInBowl AND cmIsRunning(interface.cmd.speed);
	this.TON_VibratorBowlEmpty.PT := T#3s;
	this.TON_VibratorBowlEmpty();
	interface.status.vibratorBowlEmpty := this.TON_VibratorBowlEmpty.Q;

	CASE em.mode OF
		MODE_PRODUCING: producing;
		ELSE em.cmd.sc := TRUE;
	END_CASE

	alarm;

	em();

	flapControl;
	beltControl;

	this.RTInfo_0.enable := TRUE;
	this.RTInfo_0();

	interface.status.state := em.state;
	interface.status.mode := em.mode;
	interface.status.beltFeederEmpty := this.hw.di_levelSensorBelt;

	recipe.onTime := MAX(10,recipe.onTime);
	recipe.offTime := MAX(10,recipe.offTime);

	// copy the recipe data
	CASE interface.cmd.copyRecipe OF

		COPY_RECIPE_NEXT_TO_WORKING:
			this.hmi.recipe 			:= this.hmi.recipeCurrent;
			gRecipe.cmd.save 			:= TRUE;
			interface.cmd.copyRecipe 	:= COPY_RECIPE_NONE;

			// Hardcode low filling for some elements. Ex. stalk, glass window and visor:
			IF elementNeedsLowFilling(gMainInterface.status.itemTypeId) THEN
				// Set low filling parameters
				recipe.startDelay := 3000;
				recipe.stopDelay := 10;
				recipe.onTime := 200;
				recipe.offTime := 2000;
				recipe.levelSensor := LEVEL_SENSOR_LOW;
			ELSE
				// Set default filling parameters
				recipe.startDelay := 500;
				recipe.stopDelay := 10;
				recipe.onTime := 1000;
				recipe.offTime := 300;
			END_IF

		COPY_RECIPE_SANDBOX_TO_NEXT:
			interface.cmd.copyRecipe 	:= COPY_RECIPE_NONE;

	END_CASE

	IF gRecipe.status.doCheckForChanges AND NOT this.oldCheckChangesRecipe THEN
		this.MpRecipeRegPar_Recipe.Enable := TRUE;
		this.MpRecipeRegPar_RecipeCurrent.Enable := TRUE;

		IF gRecipe.status.loaded AND NOT this.oldLoadedRecipe THEN
			// Initial program load. Set old=new to avoid saving just after a load (makes no sense)
			this.recipeOld := this.hmi.recipe;
		END_IF
		this.oldLoadedRecipe := gRecipe.status.loaded;

		IF NOT gRecipe.cmd.save AND gRecipe.status.loaded AND (brsmemcmp(ADR(this.hmi.recipe),ADR(this.recipeOld),SIZEOF(this.recipeOld)) <> 0) THEN
			gRecipe.cmd.save := TRUE;
			this.recipeOld := this.hmi.recipe;
		END_IF

	END_IF
	this.MpRecipeRegPar_Recipe(MpLink := ADR(mpRecipe), PVName := ADR(this.recipeName), Category := ADR('recipe'));
	this.MpRecipeRegPar_RecipeCurrent(MpLink := ADR(mpRecipeCurrent), PVName := ADR(this.recipeNameCurrent), Category := ADR('recipeCurrent'));
	this.oldCheckChangesRecipe := gRecipe.status.doCheckForChanges;

	IF gConfig.status.doCheckForChanges AND NOT this.oldCheckChangesConfig THEN
		this.MpRecipeRegPar_Config.Enable := TRUE;

		IF gConfig.status.loaded AND NOT this.oldLoaded THEN
			// Initial program load. Set old=new to avoid saving just after a load (makes no sense)
			this.configOld := this.hmi.config;
		END_IF
		this.oldLoaded := gConfig.status.loaded;

		IF NOT gConfig.cmd.save AND gConfig.status.loaded AND (brsmemcmp(ADR(this.hmi.config),ADR(this.configOld),SIZEOF(this.configOld)) <> 0) THEN
			gConfig.cmd.save := TRUE;
			this.configOld := this.hmi.config;
		END_IF

	END_IF
	this.MpRecipeRegPar_Config(MpLink := ADR(mpRecipe), PVName := ADR(this.configName), Category := ADR('config'));
	this.oldCheckChangesConfig := gConfig.status.doCheckForChanges;

	IF gConfig.status.factoryReset[0] THEN
		gConfig.status.factoryReset[0] := FALSE;
		// Factory reset all parameters:
		recipe.offTime := 300;
		recipe.onTime := 1000;
		recipe.startDelay := 500;
		recipe.stopDelay := 10;
	END_IF

	// FAT Level sensor test
	IF interface.cmd.levelSensorTestActive THEN
		this.hw.do_levelSensorInBowlLow 	:= interface.cmd.setLevelSensor[0];
		this.hw.do_levelSensorInBowlMedium 	:= interface.cmd.setLevelSensor[1];
		this.hw.do_levelSensorInBowlHigh 	:= interface.cmd.setLevelSensor[2];
		interface.status.levelSensorReceiverInBowl := this.hw.di_levelSensorInBowl;
	END_IF

	// FAT FLAP TEST:
	IF gFeederInterface.cmd.startFlapTest THEN
		CASE this.state OF

			0:
				IF gFeederInterface.cmd.startFlapTest THEN
					gFeederInterface.status.flapTest := TEST_NOT_DONE;
					this.state := 10;
				END_IF

			10:
				//	em.description := 'Flap opening';

				this.flap.cmd.open := TRUE;

				IF this.flap.state = FEEDER_FLAP_OPENED THEN
					this.flap.cmd.open := FALSE;
					this.state := 20;
				END_IF

			20:
				//em.description := 'flap closing and run belt forward';

				this.flap.cmd.close := TRUE;

				IF this.flap.state = FEEDER_FLAP_CLOSED THEN
					this.flap.cmd.close :=  FALSE;
					gFeederInterface.cmd.startFlapTest := FALSE;
					this.testTimeout(IN:=FALSE);
					gFeederInterface.status.flapTest := TEST_OK;
					this.state := 0;
				END_IF

		END_CASE
		this.testTimeout.IN := TRUE;
		this.testTimeout.PT := T#20s;
		this.testTimeout();
		IF this.testTimeout.Q THEN
			this.flap.cmd.open := FALSE;
			this.flap.cmd.close := TRUE;
			IF this.flap.state = FEEDER_FLAP_CLOSED THEN
				this.flap.cmd.close :=  FALSE;
				this.state := 0;
				this.testTimeout(IN:=FALSE);
				gFeederInterface.cmd.startFlapTest := FALSE;
				gFeederInterface.status.flapTest := TEST_NOT_OK;
			END_IF

		END_IF
		IF this.hmi.cmd.stopFlapTest THEN
			this.flap.cmd.open := FALSE;
			this.testTimeout(IN:=FALSE);
			this.flap.cmd.close := TRUE;
			IF this.flap.state = FEEDER_FLAP_CLOSED THEN
				this.flap.cmd.close :=  FALSE;
				this.state := 0;
				this.hmi.cmd.stopFlapTest := FALSE;
				gFeederInterface.cmd.startFlapTest := FALSE;
				gFeederInterface.status.flapTest := TEST_NOT_OK;
			END_IF

		END_IF

	END_IF

END_PROGRAM

PROGRAM _EXIT

	this.MpRecipeRegPar_Recipe(Enable := FALSE);
	this.MpRecipeRegPar_Config(Enable := FALSE);
	this.MpRecipeRegPar_RecipeCurrent(Enable := FALSE);

END_PROGRAM
```

#### setupPointers.st
```iecst
ACTION setupPointers:
	recipe ACCESS ADR(this.hmi.recipe);
	config ACCESS ADR(this.hmi.config);
	interface ACCESS ADR(gFeederInterface);

END_ACTION
```

#### local.typ - Local data types
```iecst
TYPE
	config_feeder_typ : 	STRUCT
		alarmLowLevelTime : UDINT := 15000000;
		overCurrentProtectTime : TIME := T#400ms;
		maxOpenCloseTime : TIME := T#8s;
		experimentalRefilling : BOOL;
	END_STRUCT;
	flap_typ : 	STRUCT
		state : flap_state_typ;
		internal : flap_internal_typ;
		cmd : flap_cmd_typ;
	END_STRUCT;
	flap_cmd_typ : 	STRUCT
		open : BOOL;
		close : BOOL;
	END_STRUCT;
	flap_internal_typ : 	STRUCT
		TON_maxCloseTime : TON;
		TON_maxOpenTime : TON;
		TON_delaySwitch : TON;
		TON_overCurrentProtect : TON;
		oldState : flap_state_typ;
	END_STRUCT;
	flap_state_typ :
		(
		FEEDER_FLAP_IDLE := 0,
		FEEDER_FLAP_OPENING := 1,
		FEEDER_FLAP_OPENED := 2,
		FEEDER_FLAP_CLOSING := 3,
		FEEDER_FLAP_CLOSED := 4
		);
	belt_typ : 	STRUCT
		state : belt_state_typ;
		internal : belt_internal_typ;
		cmd : belt_cmd_typ;
	END_STRUCT;
	belt_cmd_typ : 	STRUCT
		forwards : BOOL;
		backwards : BOOL;
	END_STRUCT;
	belt_state_typ :
		(
		FEEDER_BELT_IDLE := 0,
		FEEDER_BELT_FORWARDS := 1,
		FEEDER_BELT_BACKWARDS := 2
		);
	belt_internal_typ : 	STRUCT
		TON_delaySwitch : TON;
		oldState : flap_state_typ;
	END_STRUCT;
	hmi_cmd_typ : 	STRUCT
		stop : BOOL;
		empty : BOOL;
		confirmEmpty : BOOL; (*If user press confirm button before BF has been emptied, BF should exit "STATE_COMPLETING" and be ready for production. Otherwise BF will be stuck*)
		enable : BOOL := TRUE; (*Enable/disable BF*)
		forceForwards : BOOL;
		forceBackwards : BOOL;
		expFillingVisible : BOOL;
		stopFlapTest : BOOL;
	END_STRUCT;
	hmi_status_typ : 	STRUCT
		running : BOOL;
		flapOpen : BOOL;
		flapClose : BOOL;
	END_STRUCT;
	hmi_typ : 	STRUCT
		status : hmi_status_typ;
		cmd : hmi_cmd_typ;
		config : config_feeder_typ;
		recipe : recipe_feeder_typ;
		recipeCurrent : recipe_feeder_typ;
	END_STRUCT;
	local_alarm_typ : 	STRUCT
		lowLevel : gAlarm_struct_typ;
		boxMissing : gAlarm_struct_typ;
		cannotCloseFlap : gAlarm_struct_typ;
		cannotOpenFlap : gAlarm_struct_typ;
		beltFeederEmpty : gAlarm_struct_typ;
		TON_timeout : TON := (PT:=T#20s);
	END_STRUCT;
	local_hw_typ : 	STRUCT
		di_levelSensorBelt : BOOL; (*Signal name: DI_BF_LEV
PJ95: BF_S
Connector: DI.20
Description: Signal from belt feeder BF91. ”1” indicates level transmitter is activated*)
		di_boxIsReadyAtFlap : BOOL; (*Signal name: DI_BF_BOX
PJ95: BF_S
Connector: DI.21
Description: Signal form belt feeder BF91. ”1” indicates a box is ready at the belt feeder empty flap*)
		di_flapIsClosed : BOOL; (*Signal name: DI_BF_FC
PJ95: BF_S
Connector: DI.22
Description: Signal from belt feeder BF91. ”1” indicates empty flap is closed*)
		di_flapIsOpen : BOOL; (*Signal name: DI_BF_FO
PJ95: BF_S
Connector: DI.23
Description: Signal from belt feeder BF91. ”0” indicates empty flap is open*)
		do_beltForwards : BOOL; (*Signal name: DO_BF_FW
PJ95: BF_P
Connector: DO.20
Description: Signal to belt feeder: “1” means belt is driven forward if a BF91 is connected (DI_BF_91 is activated). “1” means power supply activated if a BF87 is connected (DI_BF_91 is not activated)*)
		do_beltBackwards : BOOL; (*Signal name: DO_BF_BW
PJ95: BF_P
Connector: DO.21
Description: Signal to belt feeder: “1” means belt is driven backwards if a BF91 is connected (DI_BF_91 is activated). “1” means belt is activated if a BF87 is connected (DI_BF_91 is not activated)*)
		di_levelSensorInBowl : BOOL; (*Signal name: DI_CF_LEV
PJ95: B100
Connector: DI.04
Description: Signal from CF. “0” indicates level receiver in CF is low*)
		do_levelSensorInBowlLow : BOOL; (*Signal name: DO_CF_LL
PJ95: B101
Connector: DO.01
Description: Signal to CF. “1” means low level transmitter is activated*)
		do_levelSensorInBowlMedium : BOOL; (*Signal name: DO_CF_LM
PJ95: B102
Connector: DO.02
Description: Signal to CF. “1” means medium level transmitter is activated*)
		do_levelSensorInBowlHigh : BOOL; (*Signal name: DO_CF_LH
PJ95: B103
Connector: DO.03
Description: Signal to CF. “1” means high level transmitter is activated*)
		do_flapOpen : BOOL;
		do_flapClose : BOOL;
	END_STRUCT;
	local_typ : 	STRUCT
		belt : belt_typ;
		flap : flap_typ;
		alarm : local_alarm_typ;
		hw : local_hw_typ;
		configName : STRING[80];
		recipeName : STRING[80];
		recipeNameCurrent : STRING[80];
		MpRecipeRegPar_Config : MpRecipeRegPar;
		MpRecipeRegPar_Recipe : MpRecipeRegPar;
		MpRecipeRegPar_RecipeCurrent : MpRecipeRegPar;
		hmi : hmi_typ;
		configOld : config_feeder_typ;
		recipeOld : recipe_feeder_typ;
		TON_lowLevel : TON;
		TON_timeout : TON := (PT:=T#10s);
		oldCheckChangesConfig : BOOL;
		oldCheckChangesRecipe : BOOL;
		oldLoaded : BOOL;
		oldLoadedRecipe : BOOL;
		lowLevelTime : UDINT;
		TON_VibratorBowlEmpty : TON;
		RTInfo_0 : RTInfo;
		startCounter : UDINT;
		onCounter : UDINT;
		offCounter : UDINT;
		stopCounter : UDINT;
		TON_startDelay : TON;
		state : USINT;
		testTimeout : TON;
	END_STRUCT;
	recipe_feeder_typ : 	STRUCT
		levelSensor : INT; (*10=low, 11=middle, 12=high*)
		startDelay : INT := 500; (*ms*)
		stopDelay : INT := 10; (*ms*)
		onTime : INT := 1000; (*ms*)
		offTime : INT := 300; (*ms*)
	END_STRUCT;
END_TYPE
```

#### local.var - Local variables
```iecst
VAR
	interface : REFERENCE TO gFeederInterface_typ;
	this : {REDUND_UNREPLICABLE} local_typ;
	em : {REDUND_UNREPLICABLE} brdkEM;
	recipe : REFERENCE TO recipe_feeder_typ;
	config : REFERENCE TO config_feeder_typ;
END_VAR
VAR CONSTANT
	LEVEL_SENSOR_LOW : USINT := 0;
	LEVEL_SENSOR_MEDIUM : USINT := 1;
	LEVEL_SENSOR_HIGH : USINT := 2;
END_VAR
VAR RETAIN
	flapClosing : BOOL;
	flapOpening : BOOL;
END_VAR
```

#### LocalFunctions.fun
```iecst
FUNCTION cmIsRunning : BOOL
	VAR_INPUT
		speed : LEGO_SPEED_ENUM;
	END_VAR
END_FUNCTION

FUNCTION elementNeedsLowFilling : BOOL
	VAR_INPUT
		DesignId : DINT;
	END_VAR
END_FUNCTION
```

#### LocalFunctions.st
```iecst
(* TODO: Add your comment here *)
FUNCTION cmIsRunning

	cmIsRunning := speed = lego_speed_counting OR speed = lego_speed_wait;

END_FUNCTION

FUNCTION elementNeedsLowFilling

	elementNeedsLowFilling := DesignId = 3741 OR DesignId = 24855 OR DesignId = 2447 OR DesignId = 35334 OR DesignId = 35315 OR DesignId = 35287 OR DesignId = 2586 OR DesignId = 19119;

END_FUNCTION
```

### feederGlobal.typ
```iecst
TYPE
	gFeederInterface_typ : 	STRUCT
		cmd : gFeederInterface_cmd_typ;
		status : gFeederInterface_status_typ;
	END_STRUCT;
	gFeederInterface_cmd_typ : 	STRUCT
		speed : LEGO_SPEED_ENUM;
		stop : BOOL;
		start : BOOL;
		copyRecipe : copy_recipe_command_typ;
		empty : BOOL; (*OpcUA empty cmd in main needs this to empty feeder*)
		setLevelSensor : ARRAY[0..2]OF BOOL; (*0: Low, 1: Medium, 2: High*)
		startFlapTest : BOOL;
		levelSensorTestActive : BOOL;
	END_STRUCT;
	gFeederInterface_status_typ : 	STRUCT
		running : BOOL; (*The belt is moving*)
		count : UDINT; (*Count of bricks that has passed through the photo sensor*)
		mode : DINT;
		state : brdk_em_states_typ;
		beltFeederEmpty : BOOL;
		vibratorBowlEmpty : BOOL;
		levelSensorReceiverInBowl : BOOL;
		flapTest : testResult_enum;
	END_STRUCT;
END_TYPE
```

### feederGlobal.var
```iecst
VAR
	gFeederInterface : gFeederInterface_typ;
END_VAR
```

### Program Logical/modules/main/main (IEC)

#### producing.st
```iecst
ACTION producing:

	CASE em.state OF

		STATE_RESETTING:
			this.hw.do_wo_ON	:= TRUE;
			this.reteach := FALSE;
			em.cmd.sc := TRUE;

		STATE_IDLE:

			em.description := 'Waiting for operator confirm of mechanical settings';

			IF this.newRecipeLoaded AND NOT interface.status.emptying THEN
			//	this.hmi.openConfirmDialog := TRUE;
			//	IF this.hmi.cmd.confirm THEN
			//		this.hmi.openConfirmDialog := FALSE;
			em.cmd.start := em.cmd.sc := TRUE;
			this.newRecipeLoaded := FALSE;
			//	END_IF
			ELSE
				em.cmd.start := TRUE;
			END_IF

			em.cmd.sc := TRUE;

		STATE_STARTING:

			em.description := 'Waiting for sub modules to finish starting';

			interface.status.machineFirstStart := TRUE;
			interface.status.feederStart := TRUE;
			gRecipe.status.newRecipeLoaded := brdkStrCmp(ADR(recipe.itemNumber),ADR(this.oldItemNumber)) <> 0;
			this.oldItemNumber := recipe.itemNumber;
			// If user will empty machine while capcon is teaching
			IF this.hmi.cmd.empty = 1 OR gMainInterface.line.empty THEN
				gCapconInterface.cmd.emptyWhileTeaching := TRUE;
				this.hmi.cmd.redoTeaching := TRUE;
			END_IF

			em.cmd.sc := TRUE;

		STATE_EXECUTE:
			interface.status.feederStart := (this.hmi.cmd.start OR interface.line.start);

			IF (this.hmi.cmd.empty = 1 OR gMainInterface.line.empty OR interface.status.emptying OR gCapconInterface.cmd.emptyWhileTeaching) THEN
				interface.status.emptying := TRUE;
				IF interface.cmd.wingReadyToEmpty THEN
					this.alarm.cantEmptyNeedCassette.active := FALSE;
					gCapconInterface.cmd.emptyWhileTeaching := FALSE;
					em.cmd.complete := TRUE;
				ELSE
					this.alarm.cantEmptyNeedCassette.active := TRUE;
				END_IF
			END_IF

			em.cmd.sc := TRUE;

		STATE_SUSPENDED:

			em.description := 'Wing ready to receive drop';

			em.cmd.start := NOT interface.cmd.capconWaiting OR USINT_TO_BOOL(this.hmi.cmd.empty) OR gMainInterface.line.empty;
			em.cmd.sc := TRUE;

		STATE_COMPLETING:

			CASE em.substate OF

				0:
					gWingInterface.cmd.emptyStart := TRUE;

					em.substate := 10;

				10:
					interface.status.emptying := TRUE;
					interface.status.feederStop := FALSE;
					interface.status.feederStart := FALSE;

					em.description := 'wait for machine to be empty confirm';

					IF this.hmi.cmd.confirm OR this.hmi.cmd.stop THEN // In some very odd situation it happened that the dialog with "confirm empty" didnt show and operator couldn't stop machine. Not the stop button will also stop the empty routine.
						this.hmi.cmd.confirm := FALSE;
						interface.line.emptyMode := FALSE;
						interface.line.empty := FALSE;
						hmiEmptyMode := FALSE;
						interface.status.emptying := FALSE;
						gWingInterface.cmd.confirmEmpty := TRUE;
						em.substate := 20;
					END_IF

				20:
					em.description := 'waiting for empty to finish';

					interface.status.doCalibrate := TRUE;

					em.cmd.sc := TRUE;

			END_CASE

		STATE_COMPLETE:

			gCapconInterface.cmd.reTeach := TRUE;
			interface.status.doCalibrate := FALSE;

			em.cmd.stop := em.cmd.sc := TRUE;

		STATE_STOPPING,STATE_ABORTING:

			interface.status.feederStart := FALSE;
			interface.status.feederStop := TRUE;
			this.hmi.cmd.confirm := FALSE;
			em.cmd.sc := TRUE;

		STATE_STOPPED:

			em.description	:= 'waiting for cmd';

			IF gWingInterface.status.stepperWUConnected THEN
				em.cmd.reset := (this.hw.di_stepperWUExecute[0] OR this.hw.di_stepperWUExecute[1]) AND (this.reteach OR this.hmi.cmd.start OR interface.line.start OR USINT_TO_BOOL(this.hmi.cmd.empty));
			ELSE
				em.cmd.reset := this.reteach OR this.hmi.cmd.start OR USINT_TO_BOOL(this.hmi.cmd.empty) OR interface.line.start;
			END_IF

			interface.status.emptying := USINT_TO_BOOL(this.hmi.cmd.empty);

			interface.status.feederStop := this.hmi.cmd.stop;
			interface.status.feederStart := FALSE;

			IF gWingInterface.cmd.changeMode THEN
				gWingInterface.cmd.changeMode := FALSE;
				em.mode := MODE_MANUAL;
			END_IF

		//	this.hmi.openConfirmDialog := FALSE;

			this.hmi.cmd.stop := FALSE;

			FOR i := 0 TO 20 BY 1 DO
				IF gMainInterface.cmd.activateCalibrateMode[i] THEN
					em.mode := MODE_CALIBRATING;
				END_IF

			END_FOR

			em.cmd.sc := TRUE;

		STATE_ABORTED:

			IF NOT MpAlarmXCheckReaction(mpAlarmXCore,'abortMain') THEN
				em.cmd.clear := em.cmd.sc := TRUE;
			END_IF

		STATE_CLEARING:

			brsmemset(ADR(this.alarm), 0, SIZEOF(this.alarm));
			// Alarm texts
			this.alarm.cantEmptyNeedCassette.name := 'cantEmptyNeedCassette';
			this.alarm.opcuaMethodError.name := 'opcuaMethodError';
			this.alarm.KA10.name := 'KA10ModuleError';
			this.alarm.KA11.name := 'KA11ModuleError';
			this.alarm.KA12.name := 'KA12ModuleError';
			this.alarm.KA13.name := 'KA13ModuleError';
			this.alarm.KA14.name := 'KA14ModuleError';
			this.alarm.KA15.name := 'KA15ModuleError';
			this.alarm.KA16.name := 'KA16ModuleError';
			this.alarm.KA17.name := 'KA17ModuleError';
			this.alarm.KA18.name := 'KA18ModuleError';
			this.alarm.KA19.name := 'KA19ModuleError';

			this.TON_clearing(IN := TRUE, PT := T#1s);
			gBottomFlapInterface.status.neighbourDisappeared := FALSE;
			this.hw.do_clearWU	:= TRUE;
			IF this.TON_clearing.Q THEN
				this.hw.do_clearWU	:= FALSE;
				this.TON_clearing(IN := FALSE);
				em.cmd.sc := TRUE;
			END_IF

		ELSE

			em.cmd.sc := TRUE;

	END_CASE

	this.hw.do_wo_ON := em.state <> STATE_STOPPED AND em.state <> STATE_COMPLETE AND em.state <> STATE_ABORTED AND NOT gWingInterface.status.wingEmpty;

END_ACTION
```

#### calibrating.st
```iecst
ACTION calibrating:

	CASE em.state OF

		STATE_STOPPED:

			em.mode := MODE_PRODUCING;

			IF NOT this.hmi.cmd.stop THEN

				FOR i := 0 TO 20 BY 1 DO
					IF gMainInterface.cmd.activateCalibrateMode[i] THEN
						em.mode := MODE_CALIBRATING;
					END_IF

				END_FOR

				IF 	em.mode = MODE_CALIBRATING THEN
					em.cmd.reset := TRUE;
				END_IF
			ELSE
				this.hmi.cmd.stop := FALSE;
			END_IF

			em.cmd.sc := TRUE;

		STATE_IDLE:

			em.cmd.start := em.cmd.sc := TRUE;

		STATE_EXECUTE:

			em.cmd.sc := TRUE;
			em.cmd.stop := TRUE;
			FOR i := 0 TO 20 BY 1 DO
				IF gMainInterface.cmd.activateCalibrateMode[i] THEN
					em.cmd.stop := FALSE;
				END_IF

			END_FOR

		STATE_ABORTED:

			IF NOT MpAlarmXCheckReaction(mpAlarmXCore,'abortMain') THEN
				em.cmd.clear := em.cmd.sc := TRUE;
			END_IF

		STATE_CLEARING:

			brsmemset(ADR(this.alarm), 0, SIZEOF(this.alarm));
			// Alarm texts
			this.alarm.cantEmptyNeedCassette.name := 'cantEmptyNeedCassette';
			this.alarm.opcuaMethodError.name := 'opcuaMethodError';
			this.alarm.KA10.name := 'KA10ModuleError';
			this.alarm.KA11.name := 'KA11ModuleError';
			this.alarm.KA12.name := 'KA12ModuleError';
			this.alarm.KA13.name := 'KA13ModuleError';
			this.alarm.KA14.name := 'KA14ModuleError';
			this.alarm.KA15.name := 'KA15ModuleError';
			this.alarm.KA16.name := 'KA16ModuleError';
			this.alarm.KA17.name := 'KA17ModuleError';
			this.alarm.KA18.name := 'KA18ModuleError';
			this.alarm.KA19.name := 'KA19ModuleError';
			em.cmd.sc := TRUE;
		ELSE

			em.cmd.sc := TRUE;

	END_CASE

END_ACTION
```

#### testing.st
```iecst
ACTION testing:

	CASE em.state OF

		STATE_STOPPED:

			IF gWingInterface.cmd.changeMode THEN
				gWingInterface.cmd.changeMode := FALSE;
				em.mode := MODE_PRODUCING;
			END_IF
			em.cmd.sc := TRUE;

		STATE_IDLE:

			em.cmd.start := em.cmd.sc := TRUE;

		STATE_EXECUTE:

			em.cmd.sc := TRUE;

		STATE_ABORTED:

			IF NOT MpAlarmXCheckReaction(mpAlarmXCore,'abortMain') THEN
				em.cmd.clear := em.cmd.sc := TRUE;
			END_IF

		STATE_CLEARING:

			brsmemset(ADR(this.alarm), 0, SIZEOF(this.alarm));
			// Alarm texts
			this.alarm.cantEmptyNeedCassette.name := 'cantEmptyNeedCassette';
			this.alarm.opcuaMethodError.name := 'opcuaMethodError';
			this.alarm.KA10.name := 'KA10ModuleError';
			this.alarm.KA11.name := 'KA11ModuleError';
			this.alarm.KA12.name := 'KA12ModuleError';
			this.alarm.KA13.name := 'KA13ModuleError';
			this.alarm.KA14.name := 'KA14ModuleError';
			this.alarm.KA15.name := 'KA15ModuleError';
			this.alarm.KA16.name := 'KA16ModuleError';
			this.alarm.KA17.name := 'KA17ModuleError';
			this.alarm.KA18.name := 'KA18ModuleError';
			this.alarm.KA19.name := 'KA19ModuleError';
			em.cmd.sc := TRUE;
		ELSE

			em.cmd.sc := TRUE;

	END_CASE

END_ACTION
```

#### alarm.st
```iecst
ACTION alarm:

	this.TON_0.IN := TRUE;
	this.TON_0.PT := T#200ms; // only check all these alarms every 200ms.
	this.TON_0();

	IF this.TON_0.Q THEN
		this.TON_0.IN := FALSE;
		this.TON_0();
		this.updateStatus := TRUE; // signal to update status.

		interface.status.machineType := config.machineType;
		IF gBeltInterface.cmd.setDirection THEN
			gBeltInterface.cmd.setDirection := FALSE;
			config.machineType := gBeltInterface.parameter.direction;
		END_IF
		// Can't empty machine because we need a cassette

		IF this.alarm.cantEmptyNeedCassette.active AND NOT this.alarm.cantEmptyNeedCassette.oldActive THEN
			this.alarm.cantEmptyNeedCassette.instanceID := MpAlarmXSet(mpAlarmXCore, this.alarm.cantEmptyNeedCassette.name);
		END_IF

		// reaction. Acknowledge automatically if falling edge on alarm
		IF NOT this.alarm.cantEmptyNeedCassette.active AND this.alarm.cantEmptyNeedCassette.oldActive THEN
			MpAlarmXAcknowledgeID(mpAlarmXCore, this.alarm.cantEmptyNeedCassette.instanceID);
		END_IF
		this.alarm.cantEmptyNeedCassette.oldActive := this.alarm.cantEmptyNeedCassette.active;

		// If brdkOPCUAMethodOperate is in error (then the machine can't recieve commands from gateway)

		this.alarm.opcuaMethodError.active := brdkOPCUAMethodOperate_SetMode.state = BRDK_OPCUA_METHOD_ERROR;
		IF this.alarm.opcuaMethodError.active AND NOT this.alarm.opcuaMethodError.oldActive THEN
			this.alarm.opcuaMethodError.instanceID := MpAlarmXSet(mpAlarmXCore, this.alarm.opcuaMethodError.name);
		END_IF
		// Reaction. Acknoledge if falling edge on alarm
		IF NOT this.alarm.opcuaMethodError.active AND this.alarm.opcuaMethodError.oldActive THEN
			MpAlarmXAcknowledgeID(mpAlarmXCore, this.alarm.opcuaMethodError.instanceID);
		END_IF
		this.alarm.opcuaMethodError.oldActive := this.alarm.opcuaMethodError.active;

		// IO Link module alarm ( Brick sensor belt and leve bowl)

		IF NOT this.alarm.KA10.active AND this.alarm.KA10.oldActive THEN
			this.alarm.KA10.instanceID := MpAlarmXSet(mpAlarmXCore, this.alarm.KA10.name);
		END_IF
		this.alarm.KA10.oldActive := this.alarm.KA10.active;

		// Digital Outputs 1 module alarm (bowl level and becon)

		IF NOT this.alarm.KA11.active AND this.alarm.KA11.oldActive THEN
			this.alarm.KA11.instanceID := MpAlarmXSet(mpAlarmXCore, this.alarm.KA11.name);
		END_IF
		this.alarm.KA11.oldActive := this.alarm.KA11.active;

		// Analog Inputs module alarm (Capcon)

		IF NOT this.alarm.KA12.active AND this.alarm.KA12.oldActive THEN
			this.alarm.KA12.instanceID := MpAlarmXSet(mpAlarmXCore, this.alarm.KA12.name);
		END_IF
		this.alarm.KA12.oldActive := this.alarm.KA12.active;

		// Potential Distributor module alarm (GND)

		IF NOT this.alarm.KA13.active AND this.alarm.KA13.oldActive THEN
			this.alarm.KA13.instanceID := MpAlarmXSet(mpAlarmXCore, this.alarm.KA13.name);
		END_IF
		this.alarm.KA13.oldActive := this.alarm.KA13.active;

		// Digital Inputs 1 module alarm (Wing flaps change)

		IF NOT this.alarm.KA14.active AND this.alarm.KA14.oldActive THEN
			this.alarm.KA14.instanceID := MpAlarmXSet(mpAlarmXCore, this.alarm.KA14.name);
		END_IF
		this.alarm.KA14.oldActive := this.alarm.KA14.active;

		// Digital Inputs 2 module alarm (Wing and Cassette)

		IF NOT this.alarm.KA15.active AND this.alarm.KA15.oldActive THEN
			this.alarm.KA15.instanceID := MpAlarmXSet(mpAlarmXCore, this.alarm.KA15.name);
		END_IF
		this.alarm.KA15.oldActive := this.alarm.KA15.active;

		// Digital Outputs 2 module alarm (Wing and Cassette)

		IF NOT this.alarm.KA16.active AND this.alarm.KA16.oldActive THEN
			this.alarm.KA16.instanceID := MpAlarmXSet(mpAlarmXCore, this.alarm.KA16.name);
		END_IF
		this.alarm.KA16.oldActive := this.alarm.KA16.active;

		// Digital Outputs 3 module alarm (Feeder and bottom flap)

		IF NOT this.alarm.KA17.active AND this.alarm.KA17.oldActive THEN
			this.alarm.KA17.instanceID := MpAlarmXSet(mpAlarmXCore, this.alarm.KA17.name);
		END_IF
		this.alarm.KA17.oldActive := this.alarm.KA17.active;

		// Digital input 3 module alarm (Feeder)

		IF NOT this.alarm.KA18.active AND this.alarm.KA18.oldActive THEN
			this.alarm.KA18.instanceID := MpAlarmXSet(mpAlarmXCore, this.alarm.KA18.name);
		END_IF
		this.alarm.KA18.oldActive := this.alarm.KA18.active;

		// Digital Outputs 4 module alarm (Flaps)

		IF NOT this.alarm.KA19.active AND this.alarm.KA19.oldActive THEN
			this.alarm.KA19.instanceID := MpAlarmXSet(mpAlarmXCore, this.alarm.KA19.name);
		END_IF
		this.alarm.KA19.oldActive := this.alarm.KA19.active;

		(*	Comment out and create alarms in alarmX mp file when all machines are equal!
		// Module ok KA20
		this.alarm.KA18.name := 'KA20ModuleError';
		IF NOT this.alarm.KA20 AND this.alarm.KA20.oldActive THEN
			this.alarm.KA18.instanceID := MpAlarmXSet(mpAlarmXCore, this.alarm.KA20.name);
		END_IF
		this.alarm.KA20.oldActive := this.alarm.KA20.active;

		// Module ok KA21
		this.alarm.KA21.name := 'KA21ModuleError';
		IF NOT this.alarm.KA21 AND this.alarm.KA21.oldActive THEN
			this.alarm.KA21.instanceID := MpAlarmXSet(mpAlarmXCore, this.alarm.KA21.name);
		END_IF
		this.alarm.KA21.oldActive := this.alarm.KA21.active;

		// Module ok KA22
		this.alarm.KA22.name := 'KA22ModuleError';
		IF NOT this.alarm.KA22 AND this.alarm.KA22.oldActive THEN
			this.alarm.KA22.instanceID := MpAlarmXSet(mpAlarmXCore, this.alarm.KA22.name);
		END_IF
		this.alarm.KA22.oldActive := this.alarm.KA22.active;
	*)

		(*	now using PWM anymore
		// Digital output PWM module alarm
		this.alarm.KA20.name := 'KA20ModuleError';
		IF NOT this.alarm.KA20.active AND this.alarm.KA20.oldActive THEN
			this.alarm.KA20.instanceID := MpAlarmXSet(mpAlarmXCore, this.alarm.KA20.name);
		END_IF
		this.alarm.KA20.oldActive := this.alarm.KA20.active;
		*)

		(****************************** REACTION ******************************)
		IF em.state <> STATE_ABORTED AND em.state <> STATE_ABORTING AND em.state <> STATE_CLEARING THEN
			IF MpAlarmXCheckReaction(mpAlarmXCore,'abortMain') THEN
				em.cmd.abort := TRUE;
			END_IF
		END_IF

		IF MpAlarmXCheckReaction(mpAlarmXCore,'alarmBeaconFlash') THEN
			this.alarmBeaconFlash := TRUE;
		ELSIF MpAlarmXCheckReaction(mpAlarmXCore,'alarmBeaconFlashSlow') THEN
			this.alarmBeaconFlashSlow := TRUE;
		ELSIF MpAlarmXCheckReaction(mpAlarmXCore,'alarmBeaconOn') THEN
			this.alarmBeaconOn := TRUE;
		ELSE
			this.alarmBeaconFlash := this.alarmBeaconFlashSlow := this.alarmBeaconOn := FALSE;
		END_IF
		(**********************************************************************)

	END_IF

	// Set alarm beacon depending on multiple situations
	IF this.hmi.alarmBeaconFATTest THEN
		// FAT overwrites everyone.
		this.hw.do_alarmBeacon := TRUE;
	ELSIF this.alarmBeaconFlash THEN
		this.TOF_alarmBeaconOn(IN := this.TON_alarmBeaconOff.Q, PT := T#100ms);
		this.TON_alarmBeaconOff(IN := NOT this.TOF_alarmBeaconOn.Q, PT := T#100ms);
		this.hw.do_alarmBeacon := this.TOF_alarmBeaconOn.Q;
	ELSIF this.alarmBeaconFlashSlow THEN
		this.TOF_alarmBeaconOn(IN := this.TON_alarmBeaconOff.Q, PT := T#250ms);
		this.TON_alarmBeaconOff(IN := NOT this.TOF_alarmBeaconOn.Q, PT := T#250ms);
		this.hw.do_alarmBeacon := this.TOF_alarmBeaconOn.Q;
	ELSIF this.alarmBeaconOn THEN
		this.hw.do_alarmBeacon := TRUE;
	ELSE
		this.hw.do_alarmBeacon := FALSE;
	END_IF

END_ACTION
```

#### lampCtrl.st
```iecst
ACTION lampCtrl:

	brdkOPCUAMethodOperate_LampMode();
	IF brdkOPCUAMethodOperate_LampMode.state = BRDK_OPCUA_METHOD_IS_CALLED THEN
		this.timeElapsedAfterLampCmd := 0;
		this.countBlinksLamp := 0;
		this.hw.output_lightTowerBalluff := DINT_TO_USINT(COLOR_OFF);
		TON_lamp.IN := FALSE;
		TON_lamp();
		gMachineInterface.cmd.digitalSiloCmdActive := TRUE;
		this.oldSecond := gMachineInterface.status.heartBeatFromGateway;
		brdkOPCUAMethodOperate_LampMode.finish := TRUE;
	END_IF

	IF this.hmi.startLightTowerTest THEN

		this.TON_BalluffLightTowerTest.IN := TRUE;
		this.TON_BalluffLightTowerTest.PT := T#1500ms;
		this.TON_BalluffLightTowerTest();

		IF this.TON_BalluffLightTowerTest.Q THEN
			this.TON_BalluffLightTowerTest.IN := FALSE;
			this.TON_BalluffLightTowerTest();

			this.count := this.count + 1;

			CASE this.count OF
				1: this.hw.output_lightTowerBalluff := DINT_TO_USINT(COLOR_RED);
				2: this.hw.output_lightTowerBalluff := DINT_TO_USINT(COLOR_GREEN);
				3: this.hw.output_lightTowerBalluff := DINT_TO_USINT(COLOR_BLUE);
			ELSE
				this.hw.output_lightTowerBalluff := DINT_TO_USINT(COLOR_OFF);
				this.count := 0;
				this.hmi.startLightTowerTest := FALSE;
			END_CASE

		END_IF

		IF EDGEPOS(this.hmi.startLightTowerTest) THEN
			this.count := 0;
		END_IF

		ELSIF NOT gMachineInterface.cmd.digitalSiloCmdActive THEN

			// Digital Silo Inactive - use "normal" digital output from machine.
			IF this.hw.do_alarmBeacon THEN
				this.hw.output_lightTowerBalluff := DINT_TO_USINT(COLOR_BLUE);
			ELSE
				this.hw.output_lightTowerBalluff := 0;
			END_IF

		ELSE
			// Digital silo active

			CASE lampFlash OF

				FLASH_PERMANENT:
					// Digital Silo active
					this.hw.output_lightTowerBalluff := DINT_TO_USINT(lampColor);

					// Timeout
					this.timeElapsedAfterLampCmd := this.timeElapsedAfterLampCmd + em.status.cycleTime;
					IF this.timeElapsedAfterLampCmd >= (lampTimeout*1000) THEN
						this.timeElapsedAfterLampCmd := 0;
						lampColor := COLOR_OFF;
						lampFlash := FLASH_PERMANENT;
						gMachineInterface.cmd.digitalSiloCmdActive := FALSE;
					END_IF

				FLASH_FLASH:

				// Flash interval is controlled from gateway via. UDP
				IF gMachineInterface.status.heartBeatFromGateway <> this.oldSecond THEN

					IF (gMachineInterface.status.heartBeatFromGateway MOD 2) = 0 THEN
						this.hw.output_lightTowerBalluff := DINT_TO_USINT(lampColor);
					ELSE
						this.hw.output_lightTowerBalluff := DINT_TO_USINT(COLOR_OFF);
					END_IF

				END_IF
				this.oldSecond := gMachineInterface.status.heartBeatFromGateway;

				// Timeout
				this.timeElapsedAfterLampCmd := this.timeElapsedAfterLampCmd + em.status.cycleTime;
				IF this.timeElapsedAfterLampCmd >= (lampTimeout*1000) THEN
					this.timeElapsedAfterLampCmd := 0;
					lampColor := COLOR_OFF;
					lampFlash := FLASH_PERMANENT;
					gMachineInterface.cmd.digitalSiloCmdActive := FALSE;
				END_IF

			FLASH_BLINK:

				// Blink interval is controlled from gateway via. UDP
				IF gMachineInterface.status.heartBeatFromGateway <> this.oldSecond THEN

					IF (gMachineInterface.status.heartBeatFromGateway MOD 2) = 0 THEN
						this.hw.output_lightTowerBalluff := DINT_TO_USINT(lampColor);
						this.countBlinksLamp := this.countBlinksLamp + 1;
					ELSE
						this.hw.output_lightTowerBalluff := DINT_TO_USINT(COLOR_OFF);
					END_IF

				END_IF
				this.oldSecond := gMachineInterface.status.heartBeatFromGateway;

				// lamp repeat limit
				IF this.countBlinksLamp >= lampRepeat THEN
					this.countBlinksLamp := 0;
					lampColor := COLOR_OFF;
					lampFlash := FLASH_PERMANENT;
					gMachineInterface.cmd.digitalSiloCmdActive := FALSE;
				END_IF

		END_CASE

	END_IF

END_ACTION
```

#### main.st - Init, cyclic, exit code
```iecst
PROGRAM _INIT

	gMachineType := 'CM20'; // String identifier logger system.

	em.setup.name 			:= 'main';
	em.setup.lastActivated	:= FALSE;

	// gets the task name and setup names for config and receipe types
	ST_name(0,ADR(this.configName),0);
	brdkStrCpy(ADR(this.recipeName),ADR(this.configName));
	brdkStrCpy(ADR(this.recipeNameCurrent),ADR(this.configName));
	brdkStrCat(ADR(this.configName),ADR(':this.hmi.config'));
	brdkStrCat(ADR(this.recipeName),ADR(':this.hmi.recipe'));
	brdkStrCat(ADR(this.recipeNameCurrent),ADR(':this.hmi.recipeCurrent'));

	setupPointers;

	interface.status.simulation := DiagCpuIsSimulated();
	interface.status.statusIT.Connected := TRUE;

	brdkOPCUAMethodOperate_SetMode.enable 	:= TRUE;
	brdkOPCUAMethodOperate_SetMode.name 	:= 'SetMode';
	brdkOPCUAMethodOperate_LampMode.enable := TRUE;
	brdkOPCUAMethodOperate_LampMode.name := 'LampMode';
	hmiEmptyMode;
	interface.status.statusIT.Command := 1; // STOPPED

	// Alarm texts
	this.alarm.cantEmptyNeedCassette.name := 'cantEmptyNeedCassette';
	this.alarm.opcuaMethodError.name := 'opcuaMethodError';
	this.alarm.KA10.name := 'KA10ModuleError';
	this.alarm.KA11.name := 'KA11ModuleError';
	this.alarm.KA12.name := 'KA12ModuleError';
	this.alarm.KA13.name := 'KA13ModuleError';
	this.alarm.KA14.name := 'KA14ModuleError';
	this.alarm.KA15.name := 'KA15ModuleError';
	this.alarm.KA16.name := 'KA16ModuleError';
	this.alarm.KA17.name := 'KA17ModuleError';
	this.alarm.KA18.name := 'KA18ModuleError';
	this.alarm.KA19.name := 'KA19ModuleError';

	this.hmi.cmType := 'CM20';

END_PROGRAM

PROGRAM _CYCLIC

	setupPointers;

	IF gRecipe.status.newRecipeLoaded THEN
		this.newRecipeLoaded := TRUE;
	END_IF

	// OPCUA cmds
	brdkOPCUAMethodOperate_SetMode();
	CASE brdkOPCUAMethodOperate_SetMode.state OF
		// TODO: Generate alarm if BRDK_OPCUA_ERROR occurs
		BRDK_OPCUA_METHOD_IS_CALLED:
			CASE setMode OF

				STOP:
					this.hmi.cmd.stop := TRUE;

				PRODUCTION:
					this.hmi.cmd.start := TRUE;

				PRE_EMPTY:
					interface.line.emptyMode := hmiEmptyMode := TRUE;

				PRE_EMPTY_DISABLE:
					interface.line.emptyMode := hmiEmptyMode := FALSE;

				EMPTY_OUT:
					gFeederInterface.cmd.empty := TRUE;	// cmd to feeder (feeder is not parent of main)
					this.hmi.cmd.empty := TRUE;

			END_CASE

			brdkOPCUAMethodOperate_SetMode.finish := TRUE;

	END_CASE

	// Ethernet IP cmds
	IF interface.cmd.stopEthIP AND NOT this.oldStopEthIP THEN
		// Rising edge trigger
		this.hmi.cmd.stop := TRUE;
	END_IF
	this.oldStopEthIP := interface.cmd.stopEthIP;

	IF interface.cmd.startEthIP AND NOT this.oldStartEthIP THEN
		// Rising edge trigger
		this.hmi.cmd.start := TRUE;
	END_IF
	this.oldStartEthIP := interface.cmd.startEthIP;

	IF interface.cmd.emptyEthIP AND NOT this.oldEmptyEthIP THEN
		// Rising edge trigger
		gFeederInterface.cmd.empty := TRUE;	// cmd to feeder (feeder is not parent of main)
		this.hmi.cmd.empty := TRUE;
	END_IF
	this.oldEmptyEthIP := interface.cmd.emptyEthIP;

	IF interface.cmd.emptyModeEthIP AND NOT this.oldEmptyModeEthIP THEN
		// Rising AND falling edge trigger
		interface.line.emptyMode := hmiEmptyMode := TRUE;
	END_IF
	this.oldEmptyModeEthIP := interface.cmd.emptyModeEthIP;

	interface.line.bypassCassette := interface.cmd.bypassCassetteEthIP; // bypass always dictated by line controller over ethernet ip.

	//-------------------------------- //

	// Ethernet IP status
	gEthernetIPInterface.status.stop := em.state = STATE_STOPPED;
	gEthernetIPInterface.status.start := em.state <> STATE_STOPPED;
	gEthernetIPInterface.status.empty := interface.status.emptying;
	gEthernetIPInterface.status.emptyMode := interface.line.emptyMode;
	gEthernetIPInterface.status.bypassCassette := interface.line.bypassCassette;

	em.cmd.stop := this.hmi.cmd.stop OR gRecipe.cmd.load;
	this.stopCalibration :=  em.mode = MODE_CALIBRATING AND em.state <> STATE_STOPPED;

	// Some status update for IT
	IF this.updateStatus THEN
		this.updateStatus := FALSE;
		// CM_BOOL_STATUS for gateway. 0: stopped, 1: running, 2: emptying, 3: preempty, 4: dosing
		interface.status.statusIT.BypassCassette := interface.line.bypassCassette;
		CM_BOOL_STATUS.1 := em.state=STATE_EXECUTE OR em.state=STATE_STARTING;
		CM_BOOL_STATUS.2 := em.state=STATE_COMPLETE OR em.state=STATE_COMPLETING;
		CM_BOOL_STATUS.0 := NOT CM_BOOL_STATUS.1 AND NOT CM_BOOL_STATUS.2; // If not running or emptying, then it's stopped.
		CM_BOOL_STATUS.3 := interface.line.emptyMode;
		CM_BOOL_STATUS.4 := interface.line.bypassCassette OR gCapconInterface.status.wingDosing;	// When recipe.brickCount=0 OR line command

		IF interface.line.bypassCassette THEN
			// dosing
			interface.status.statusIT.Command := 4;
		ELSIF em.state=STATE_COMPLETE OR em.state=STATE_COMPLETING THEN
			// emptying
			interface.status.statusIT.Command := 2;
		ELSIF interface.line.emptyMode THEN
			// preempty
			interface.status.statusIT.Command := 5;
		ELSE
			// Production if em is in execute/starting else stopped
			interface.status.statusIT.Command := SEL(em.state=STATE_EXECUTE OR em.state=STATE_STARTING,1,3);
		END_IF

	END_IF

	FOR i := 0 TO 20 BY 1 DO
		IF gMainInterface.cmd.activateCalibrateMode[i] THEN
			IF em.mode = MODE_PRODUCING AND em.state <> STATE_STOPPED THEN
				em.cmd.stop := TRUE;
			END_IF
			this.stopCalibration := FALSE; // do not stop calibration as one module still has calibration active
		END_IF
	END_FOR

	IF this.stopCalibration THEN
		em.cmd.stop := TRUE;
	END_IF

	interface.line.emptyMode := hmiEmptyMode; // emptyMode from hmi.

	IF this.hmi.cmd.redoTeaching AND (em.state = STATE_STARTING) THEN
		this.reteach := TRUE;
		em.cmd.stop := TRUE;
	END_IF

	CASE em.mode OF
		MODE_PRODUCING: producing;
		MODE_CALIBRATING: calibrating;
		MODE_MANUAL: testing;

		ELSE em.cmd.sc := TRUE;
	END_CASE

	interface.status.emMode := em.mode;
	interface.status.itemNumber := SEL(this.hmi.itemNumberNext <> '', recipe.itemNumber, this.hmi.itemNumberNext);
	interface.status.itemTypeId := recipe.itemTypeId;
	interface.status.machineDirection := config.machineType;
	this.hmi.showNextItemNumberLabel := this.hmi.itemNumberNext <> '';

	brdkStrMemSet(ADR(this.hmi.cmd),0,SIZEOF(this.hmi.cmd));

	alarm;
	lampCtrl;
	em();

	//Give status to wing that machine start and reset statistic
	IF em.state = STATE_EXECUTE AND em.mode = MODE_PRODUCING THEN
		interface.status.machineStart	:= TRUE;
	ELSE
		interface.status.machineStart	:= FALSE;
	END_IF

	//this.hmi.mainAborted := em.state = STATE_ABORTED;

	// copy the recipe data
	CASE interface.cmd.copyRecipe OF

		COPY_RECIPE_NEXT_TO_WORKING:
			IF interface.cmd.loadingTemplateRecipe THEN
				// Template recipe can't load itemNumber/itemTypeId
				this.itemNumber := this.hmi.recipe.itemNumber;
				this.itemTypeId := this.hmi.recipe.itemTypeId;
				this.hmi.recipe := this.hmi.recipeCurrent;
				this.hmi.recipe.itemNumber := this.itemNumber;
				this.hmi.recipe.itemTypeId := this.itemTypeId;
			ELSE
				this.hmi.recipe := this.hmi.recipeCurrent;
			END_IF
			interface.status.statusIT.ItemType := DINT_TO_UDINT(recipe.itemTypeId);
			interface.status.itemTypeId := recipe.itemTypeId;
			this.hmi.itemNumberNext := '';

			IF recipe.itemTypeId = 24855 OR recipe.itemTypeId = 3741 THEN
				// Stalk element. Put som hardcoded values for this because it is a very tricky element and we have seen some very bad values in lego DB.
				gVibratorInterface[0].cmd.putRecipeForStalkElement := gVibratorInterface[1].cmd.putRecipeForStalkElement := gBeltInterface.cmd.putRecipeForStalkElement := TRUE;
			END_IF

			gRecipe.cmd.save 			:= TRUE;
			interface.cmd.copyRecipe 	:= COPY_RECIPE_NONE;

		COPY_RECIPE_SANDBOX_TO_NEXT:
			interface.cmd.copyRecipe 	:= COPY_RECIPE_NONE;

	END_CASE

	IF gRecipe.status.doCheckForChanges AND NOT this.oldCheckChangesRecipe THEN
		this.MpRecipeRegPar_Recipe.Enable := TRUE;
		this.MpRecipeRegPar_RecipeCurrent.Enable := TRUE;
		// Update statusIT.
		interface.status.statusIT.ItemNumber := STRING_TO_UDINT(recipe.itemNumber);
		interface.status.statusIT.ItemType := DINT_TO_UDINT(recipe.itemTypeId);

		IF gRecipe.status.loaded AND NOT this.oldLoadedRecipe THEN
			// Initial program load. Set old=new to avoid saving just after a load (makes no sense)
			this.recipeOld := this.hmi.recipe;
		END_IF
		this.oldLoadedRecipe := gRecipe.status.loaded;

		IF NOT gRecipe.cmd.save AND gRecipe.status.loaded AND (brsmemcmp(ADR(this.hmi.recipe),ADR(this.recipeOld),SIZEOF(this.recipeOld)) <> 0) THEN
			gRecipe.cmd.save := TRUE;
			this.recipeOld := this.hmi.recipe;
		END_IF

	END_IF
	this.MpRecipeRegPar_Recipe(MpLink := ADR(mpRecipe), PVName := ADR(this.recipeName), Category := ADR('recipe'));
	this.MpRecipeRegPar_RecipeCurrent(MpLink := ADR(mpRecipeCurrent), PVName := ADR(this.recipeNameCurrent), Category := ADR('recipeCurrent'));
	this.oldCheckChangesRecipe := gRecipe.status.doCheckForChanges;

	IF gConfig.status.doCheckForChanges AND NOT this.oldCheckChangesConfig THEN
		this.MpRecipeRegPar_Config.Enable := TRUE;

		IF gConfig.status.loaded AND NOT this.oldLoaded THEN
			// Initial program load. Set old=new to avoid saving just after a load (makes no sense)
			this.configOld := this.hmi.config;
		END_IF
		this.oldLoaded := gConfig.status.loaded;

		IF NOT gConfig.cmd.save AND gConfig.status.loaded AND (brsmemcmp(ADR(this.hmi.config),ADR(this.configOld),SIZEOF(this.configOld)) <> 0) THEN
			gConfig.cmd.save := TRUE;
			this.configOld := this.hmi.config;
		END_IF

	END_IF
	this.MpRecipeRegPar_Config(MpLink := ADR(mpRecipe), PVName := ADR(this.configName), Category := ADR('config'));
	this.oldCheckChangesConfig := gConfig.status.doCheckForChanges;

	interface.status.state := em.state;

END_PROGRAM

PROGRAM _EXIT

	this.MpRecipeRegPar_Recipe(Enable := FALSE);
	this.MpRecipeRegPar_Config(Enable := FALSE);
	this.MpRecipeRegPar_RecipeCurrent(Enable := FALSE);
	brdkOPCUAMethodOperate_SetMode(enable:=FALSE);
	brdkOPCUAMethodOperate_LampMode(enable:=FALSE);
END_PROGRAM
```

#### setupPointers.st
```iecst
ACTION setupPointers:
	recipe ACCESS ADR(this.hmi.recipe);
	config ACCESS ADR(this.hmi.config);
	interface ACCESS ADR(gMainInterface);
END_ACTION
```

#### local.typ - Local data types
```iecst
TYPE
	set_mode_typ :
		(
		STOP := 0,
		PRODUCTION := 1,
		EMPTY_OUT := 2,
		PRE_EMPTY := 3,
		BYPASS_CASSETTE := 4,
		BYPASS_CASSETTE_DISABLE := 5,
		PRE_EMPTY_DISABLE := 6,
		EXTRA := 7
		);
	lamp_color_typ :
		(
		COLOR_OFF := 0, (*NO COLOR*)
		COLOR_GREEN := 1, (*GREEN*)
		COLOR_RED := 2, (*RED*)
		COLOR_YELLOW := 3, (*YELLOW*)
		COLOR_BLUE := 4, (*BLUE*)
		COLOR_ORANGE := 5, (*ORANGE*)
		COLOR_OWN := 6, (*OWN*)
		COLOR_WHITE := 7 (*WHITE*)
		) := COLOR_OFF;
	lamp_flash_typ :
		(
		FLASH_PERMANENT := 0,
		FLASH_FLASH := 1, (*Flash every x ms for a timeout duration*)
		FLASH_BLINK := 2 (*Blink every x ms for a count amount*)
		) := FLASH_PERMANENT;
	local_typ : 	STRUCT
		alarm : local_alarm_typ;
		hw : local_hw_typ;
		TOF_alarmBeaconOn : TOF;
		TON_alarmBeaconOff : TON;
		configName : STRING[80];
		recipeName : STRING[80];
		recipeNameCurrent : STRING[80];
		MpRecipeRegPar_Config : MpRecipeRegPar;
		MpRecipeRegPar_Recipe : MpRecipeRegPar;
		MpRecipeRegPar_RecipeCurrent : MpRecipeRegPar;
		hmi : hmi_typ;
		timeElapsed : UDINT;
		recipeOld : recipe_main_typ;
		configOld : config_main_typ;
		newRecipeLoaded : BOOL;
		interface : gMainInterface_typ;
		stopCalibration : BOOL;
		reteach : BOOL;
		oldRemoteCommand : USINT;
		oldItemNumber : STRING[100];
		itemNumber : STRING[100];
		itemTypeId : DINT;
		TON_clearing : TON;
		oldCheckChangesConfig : BOOL;
		oldCheckChangesRecipe : BOOL;
		oldLoaded : BOOL;
		oldLoadedRecipe : BOOL;
		alarmBeaconFlash : BOOL;
		alarmBeaconFlashSlow : BOOL;
		alarmBeaconOn : BOOL;
		TON_0 : TON;
		updateStatus : BOOL;
		oldStopEthIP : BOOL; (*cmd from LineController to CM20*)
		oldStartEthIP : BOOL; (*cmd from LineController to CM20*)
		oldEmptyEthIP : BOOL; (*cmd from LineController to CM20*)
		oldEmptyModeEthIP : BOOL; (*cmd from LineController to CM20*)
		oldBypassCassetteEthIP : BOOL; (*cmd from LineController to CM20*)
		timeElapsedAfterLampCmd : UDINT; (* [us]*)
		countBlinksLamp : UDINT;
		oldSecond : UDINT;
		TON_BalluffLightTowerTest : TON;
		count : USINT;
	END_STRUCT;
	hmi_cmd_typ : 	STRUCT
		empty : SINT;
		confirm : BOOL;
		stop : BOOL;
		hold : BOOL;
		start : BOOL;
		teach : BOOL;
		rejectAll : USINT;
		redoTeaching : BOOL;
	END_STRUCT;
	hmi_typ : 	STRUCT
		openConfirmDialog : BOOL;
		recipe : recipe_main_typ;
		cmd : hmi_cmd_typ;
		config : config_main_typ;
		status : USINT;
		state : STRING[80];
		stateTemp : STRING[80];
		recipeCurrent : recipe_main_typ; (*Next recipe data*)
		setMode : USINT;
		mainAborted : BOOL;
		cmType : STRING[10];
		batchId : DINT;
		imageURL : STRING[200];
		itemNumberNext : STRING[100];
		showNextItemNumberLabel : BOOL;
		startLightTowerTest : BOOL;
		alarmBeaconFATTest : BOOL;
	END_STRUCT;
	config_main_typ : 	STRUCT
		number : DINT;
		version : STRING[80];
		machineType : USINT; (*0 = left, 1 = right*)
		enableExperimental : BOOL;
	END_STRUCT;
	recipe_main_typ : 	STRUCT
		itemNumber : STRING[100]; (*Item number*)
		width : INT; (*[mm] width setting on circular vibrator*)
		height : INT; (*[mm] height setting on circular vibrator*)
		angle : INT;
		itemName : STRING[100]; (*Item name*)
		itemTypeId : DINT; (*item type/design id of brick. Unique for element design but the same for different colors/decoration*)
	END_STRUCT;
	local_hw_typ : 	STRUCT
		di_stopButton : BOOL; (*Signal name: DI_CM_STOP
PJ95: NA
Connector: B500
Description: Signal from Stop button*)
		di_startButton : BOOL; (*Signal name: DI_CM_START
PJ95: B501
Connector: NA
Description: Signal from Start button*)
		do_stopButtonIndicator : BOOL; (*Signal name: DO_CM_STOP
PJ95: B502
Connector: NA
Description: Signal to Stop button indicator*)
		do_startButtonIndicator : BOOL; (*Signal name: DO_CM_START
PJ95: B503
Connector: NA
Description: Signal to Start button indicator*)
		do_alarmBeacon : BOOL; (*Signal name: DO_CM_ALARM
PJ95: H100
Connector: DO.04
Description: Signal to alarm beacon*)
		do_wo_ON : BOOL; (*Stepper wu on command*)
		do_clearWU : BOOL;
		di_stepperWUExecute : ARRAY[0..1]OF BOOL;
		output_lightTowerBalluff : USINT;
		input_lightTowerBalluff : USINT;
	END_STRUCT;
	local_alarm_typ : 	STRUCT
		KA10 : gAlarm_struct_typ;
		KA11 : gAlarm_struct_typ;
		KA12 : gAlarm_struct_typ;
		KA13 : gAlarm_struct_typ;
		KA14 : gAlarm_struct_typ;
		KA15 : gAlarm_struct_typ;
		KA16 : gAlarm_struct_typ;
		KA17 : gAlarm_struct_typ;
		KA18 : gAlarm_struct_typ;
		KA19 : gAlarm_struct_typ;
		KA20 : gAlarm_struct_typ;
		KA21 : gAlarm_struct_typ;
		KA22 : gAlarm_struct_typ;
		cantEmptyNeedCassette : gAlarm_struct_typ;
		opcuaMethodError : gAlarm_struct_typ;
	END_STRUCT;
	remoteCmd_typ : 	STRUCT
		bypassCassette : USINT; (*Can be “On” or “Off”.  It is Bypass cassette - CM release cassette without dossing*)
		command : USINT; (*Can be “End”, “Stop”, “Start” or “Empty”.
“End” indicates that counting will cease either when the current counting process has been completed or, if the first element has not yet been counted, immediately.
“Stop” indicates that counting will stop immediately. Any count in progress will be rejected.
“Start” indicates that counting starts if the element quantity is greater than zero.
“Empty” indicates that the counting machine is to be empties for items.*)
	END_STRUCT;
END_TYPE
```

#### local.var - Local variables
```iecst
VAR
	setMode : set_mode_typ;
	lampFlash : lamp_flash_typ := FLASH_PERMANENT;
	lampColor : lamp_color_typ := COLOR_OFF;
	brdkOPCUAMethodOperate_SetMode : brdkOPCUAMethodOperate;
	brdkOPCUAMethodOperate_LampMode : brdkOPCUAMethodOperate;
	CM_BOOL_STATUS : DINT;
	i : USINT;
	interface : REFERENCE TO gMainInterface_typ;
	em : brdkEM;
	this : local_typ;
	config : REFERENCE TO config_main_typ;
	recipe : REFERENCE TO recipe_main_typ;
	hmiEmptyMode : BOOL;
	lampTimeout : UDINT := 30000; (*[ms] Time in ms*)
	lampRepeat : UDINT := 15; (*Amount of times that lamp blinks in "Blink method"*)
	lampDuration : TIME := T#1s; (*Time between flash*)
	TON_lamp : TON;
END_VAR
```

- Methods.uam (not shown)

### mainGlobal.typ
```iecst
TYPE
	gMainInterface_line_typ : 	STRUCT
		start : BOOL;
		empty : BOOL;
		emptyMode : BOOL;
		bypassCassette : BOOL;
	END_STRUCT;
	gMainInterface_typ : 	STRUCT
		cmd : gMainInterface_cmd_typ;
		status : gMainInterface_status_typ;
		line : gMainInterface_line_typ;
	END_STRUCT;
	gMainInterface_cmd_typ : 	STRUCT
		brickAtSensor : BOOL;
		capconReady : BOOL;
		state : BOOL;
		count : UDINT;
		validationTotalCount : UDINT;
		validationGoodBrick : BOOL;
		validationBadBrick : BOOL;
		capconWaiting : BOOL;
		activateCalibrateMode : ARRAY[0..20]OF BOOL;
		copyRecipe : copy_recipe_command_typ;
		wingReadyToEmpty : BOOL;
		loadingTemplateRecipe : BOOL;
		stopEthIP : BOOL; (*cmd from LineController to CM20*)
		startEthIP : BOOL; (*cmd from LineController to CM20*)
		emptyEthIP : BOOL; (*cmd from LineController to CM20*)
		emptyModeEthIP : BOOL; (*cmd from LineController to CM20*)
		bypassCassetteEthIP : BOOL; (*cmd from LineController to CM20*)
	END_STRUCT;
	gMainInterface_status_typ : 	STRUCT
		start : BOOL;
		simulation : BOOL;
		emMode : DINT;
		count : USINT;
		totalCount : UDINT;
		dpMin : REAL;
		doLinearization : BOOL;
		doCalibrate : BOOL;
		feederStop : BOOL;
		feederStart : BOOL;
		emptying : BOOL;
		machineStart : BOOL;
		machineFirstStart : BOOL; (*will be true first time main goes into STATE_STARTING*)
		itemNumber : STRING[20];
		itemTypeId : DINT; (*item type/design id of brick. Unique for element design but the same for different colors/decoration*)
		statusIT : gMainInterface_statusIT_typ;
		state : brdk_em_states_typ;
		machineDirection : USINT; (*0=left , 1=right*)
		machineType : USINT;
	END_STRUCT;
	gMainInterface_statusIT_typ : 	STRUCT
		Connected : BOOL;
		ItemNumber : UDINT;
		ItemType : UDINT;
		PortionItemCount : INT;
		SerialNo : UDINT;
		Type : INT;
		Version : STRING[20];
		BypassCassette : BOOL;
		Command : INT; (*// 0: DEACTIVATED, 1: STOPPED, 2: EMPTYING, 3: PRODUCTION, 4: DOSING *)
	END_STRUCT;
END_TYPE
```

### mainGlobal.var
```iecst
VAR
	gMainInterface : gMainInterface_typ;
END_VAR
```

### Program Logical/modules/main/vibrator/sineWaveGen (IEC)

#### Main.st - Init, cyclic, exit code
```iecst
PROGRAM _INIT

	acc.enable 	:= 	TRUE;
	acc.samples	:= 103;		// number of samples at 2kHz sample rate ~ 20 = 10ms

	FOR i:=1 TO NUM_VIBRATOR DO
		vibratorControl_0[i].vibratorType := i;	// i=0=CF , i=1=LF
		vibratorControl_0[i].pAxis := SEL(i=0,ADR(gAxisVibL),ADR(gAxisVibC));
	END_FOR

END_PROGRAM

PROGRAM _CYCLIC

	FOR i:=1 TO NUM_VIBRATOR DO

		IF local[i].readPercentFromAccelerometer OR gVibratorInterface[i].status.calibratingMode OR gVibratorInterface[i].status.forcing THEN
			local[i].percentFromAccelerometer := getPercentFromAcceleration(acc.analogVib,i,gVibratorInterface[0].status.machineType);
			gVibratorInterface[i].status.currAccelerometerPercent := local[i].percentFromAccelerometer;
			gVibratorInterface[i].status.currEstimatedPercent := vibratorControl_0[i].estimatedPercent;
			hmiAccelerometerPercent := local[i].percentFromAccelerometer;
			gVibratorInterface[i].status.currAccelerometerValue := acc.analogVib;
		END_IF

		vibratorControl_0[i].enable 		:= gVibratorInterface[i].status.powered;
		vibratorControl_0[i].amplitude		:= gVibratorInterface[i].status.vibAmplitude;
		vibratorControl_0[i].percent		:= gVibratorInterface[i].status.percent;
		vibratorControl_0[i].machineType	:= gVibratorInterface[i].status.machineType;
		vibratorControl_0[i].manualControl	:= (gVibratorInterface[i].status.calibratingMode OR gVibratorInterface[i].status.forcing) AND NOT gVibratorInterface[i].status.caliProdTest;
		vibratorControl_0[i].activateMinMax := gVibratorInterface[i].status.caliProdTest;
		vibratorControl_0[i].manualFrequency := gVibratorInterface[i].status.vibFrequency;
		vibratorControl_0[i].manualBrake	:= gVibratorInterface[i].status.calibrateBrake;
		vibratorControl_0[i].manualBoost	:= gVibratorInterface[i].status.calibrateBoost;
		vibratorControl_0[i].brakeFrequency := gVibratorInterface[i].status.brakeFrequency;
		vibratorControl_0[i].boostFrequency := gVibratorInterface[i].status.boostFrequency;
		vibratorControl_0[i].boostVelocityLow := SEL(gVibratorInterface[i].status.boostVelocityLow = 0, gVibratorInterface[i].status.boostVelocityLow, 40000);
		vibratorControl_0[i].boostVelocityHigh := SEL(gVibratorInterface[i].status.boostVelocityHigh = 0, gVibratorInterface[i].status.boostVelocityHigh, 40000);
		vibratorControl_0[i].brakeVelocity := SEL(gVibratorInterface[i].status.brakeVelocity = 0, gVibratorInterface[i].status.brakeVelocity, 40000);
		vibratorControl_0[i].boostAmplitude := gVibratorInterface[i].status.boostAmpltiude;
		vibratorControl_0[i].brakeAmplitude := gVibratorInterface[i].status.brakeAmplitude;
		vibratorControl_0[i].linearizationAmplitude := gVibratorInterface[i].status.linearizationAmplitude;
		vibratorControl_0[i].linearizationFrequencies := gVibratorInterface[i].status.linearizationFrequencies;
		vibratorControl_0[i].manualBrakeTime := LIMIT(0, gVibratorInterface[i].status.calibrateBraketime, 1);
		vibratorControl_0[i].manualBrakeAmplitudeEnd := gVibratorInterface[i].status.calibrateBrakeAmplitudeEnd;
		vibratorControl_0[i].manualBrakeFrequencyEnd := gVibratorInterface[i].status.calibrateBrakeFrequencyEnd;
		vibratorControl_0[i].currAccelerometerValue := acc.analogVib;
		vibratorControl_0[i].currAccelerometerPercent := local[i].percentFromAccelerometer;
		vibratorControl_0[i].disableBoost := gVibratorInterface[i].status.disableLFBoost;
		vibratorControl_0[i]();

		// Output mapping:
		gVibratorInterface[i].status.minAccelerationStart := vibratorControl_0[i].accelerationStart;
		gVibratorInterface[i].status.minAcceleration := vibratorControl_0[i].minAcceleration;
		gVibratorInterface[i].status.minAccelerationTime := vibratorControl_0[i].minAccelerationTime;
		gVibratorInterface[i].status.caliBoostVelocityLow := vibratorControl_0[i].caliBoostVelocityLow;
		gVibratorInterface[i].status.caliBoostVelocityHigh := vibratorControl_0[i].caliBoostVelocityHigh;
		gVibratorInterface[i].status.maxBoostPercent := vibratorControl_0[i].maxBoostPercent;
		gVibratorInterface[i].status.minBreakPercent := vibratorControl_0[i].minBreakPercent;
		gVibratorInterface[i].status.filteredAccelerometerPercent := vibratorControl_0[i].filteredAccelerometerPercent;

		// GetPhaseDifference_0.Enable := TRUE;
		GetPhaseDifference_0[i].ReferenceSignal := ABS(vibratorControl_0[i].sin_out);
		GetPhaseDifference_0[i].Signal := acc.rawVib;
		GetPhaseDifference_0[i]();

		///////////////////////////////////////////////////
		//// MANUEL CONTROL FOR FORCING AND CALIBRATION////
		///////////////////////////////////////////////////
		IF gVibratorInterface[i].cmd.readCurrentAndVoltage THEN
			local[i].MC_BR_CyclicRead_0.Enable := TRUE;
			local[i].MC_BR_CyclicRead_0.Axis := SEL(i=0,ADR(gAxisVibL),ADR(gAxisVibC));
			local[i].MC_BR_CyclicRead_0.ParID := 214;
			local[i].MC_BR_CyclicRead_0.DataType := ncPAR_TYP_REAL;
			local[i].MC_BR_CyclicRead_0.DataAddress := ADR(local[i].actCurrent);
			local[i].MC_BR_CyclicRead_0();

			local[i].MC_BR_CyclicRead_1.Enable := TRUE;
			local[i].MC_BR_CyclicRead_1.Axis := SEL(i=0,ADR(gAxisVibL),ADR(gAxisVibC));
			local[i].MC_BR_CyclicRead_1.ParID := 216;
			local[i].MC_BR_CyclicRead_1.DataType := ncPAR_TYP_REAL;
			local[i].MC_BR_CyclicRead_1.DataAddress := ADR(local[i].actVoltage);
			local[i].MC_BR_CyclicRead_1();

			local[i].time := local[i].time + CYCLE_TIME_us;
			local[i].maxPeakCurrent := MAX(ABS(local[i].actCurrent),local[i].maxPeakCurrent);
			IF local[i].time >= 100000 THEN
				// Every 0.25s send max current to vibrator task
				local[i].time := 0;
				gVibratorInterface[i].status.actCurr := local[i].maxPeakCurrent;
				local[i].maxPeakCurrent := 0;
			END_IF
		ELSE
			gVibratorInterface[i].status.actCurr := 0;
			local[i].MC_BR_CyclicRead_0(Enable:=FALSE);
			local[i].MC_BR_CyclicRead_1(Enable:=FALSE);
		END_IF

		// Max peaks
		IF gVibratorInterface[i].cmd.monitorActPeakValue THEN
			MTFilterMovingAverage_0[i].Enable := TRUE;
			MTFilterMovingAverage_0[i].In := acc.analogVib;
			MTFilterMovingAverage_0[i].WindowLength := 250;	// 400ms moving average
			MTFilterMovingAverage_0[i]();

			MTBasicsTimeDelay_0[i].Enable := TRUE;
			MTBasicsTimeDelay_0[i].DelayTime := 0.2;
			MTBasicsTimeDelay_0[i].In := gVibratorInterface[i].status.vibFrequency;;
			MTBasicsTimeDelay_0[i]();

			gVibratorInterface[i].status.maxPeakValue := MTFilterMovingAverage_0[i].Out;

		ELSIF MTFilterMovingAverage_0[i].Enable THEN
			gVibratorInterface[i].status.highestFrequency := 0;
			gVibratorInterface[i].status.highestAmplitude := 0;
			MTFilterMovingAverage_0[i].Enable := FALSE;
			MTFilterMovingAverage_0[i]();
			MTBasicsTimeDelay_0[i].Enable := FALSE;
			MTBasicsTimeDelay_0[i]();
		END_IF

		IF gVibratorInterface[i].cmd.monitorMaxPeakValue THEN

			IF gVibratorInterface[i].status.maxPeakValue > gVibratorInterface[i].status.highestAmplitude AND MTBasicsTimeDelay_0[i].Out > 0 THEN
				gVibratorInterface[i].status.highestAmplitude := gVibratorInterface[i].status.maxPeakValue;
				gVibratorInterface[i].status.highestFrequency := MTBasicsTimeDelay_0[i].Out;
			END_IF
		ELSE
			gVibratorInterface[i].status.highestAmplitude := 0;
			gVibratorInterface[i].status.highestFrequency := 0;
		END_IF
	END_FOR

	IF gVibratorInterface[0].status.isBigCF THEN
		// Big CF must use double samples because the frequency is half
		acc.samples	:= 103;		// number of samples at 2kHz sample rate ~ 1 period on accelerometer
	ELSE
		// big CF
		acc.samples	:= 53;		// number of samples at 2kHz sample rate ~ 1 period on accelerometer
	END_IF

END_PROGRAM

PROGRAM _EXIT

	FOR i:=1 TO NUM_VIBRATOR DO
		MTBasicsTimeDelay_0[i](Enable := FALSE);
		MTFilterMovingAverage_0[i](Enable := FALSE);
	END_FOR

END_PROGRAM
```

#### Types.typ - Local data types
```iecst
TYPE
	acc_typ : 	STRUCT
		samples : UINT;
		enable : BOOL; (*enable reading of acc. values*)
		actVib : REAL;
		analogVib : REAL;
		toggleBit : BOOL;
		RmsAccRaw : REAL;
		RmsVelRaw : REAL;
		PeakRaw : REAL;
		RmsRaw : REAL;
		ISO : REAL;
		rawVib : REAL;
	END_STRUCT;
	local_typ : 	STRUCT
		percentFromAccelerometer : REAL;
		MC_BR_CyclicRead_Max : MC_BR_CyclicRead;
		maxVoltage : REAL;
		MC_BR_CyclicRead_0 : MC_BR_CyclicRead;
		MC_BR_CyclicRead_1 : MC_BR_CyclicRead;
		time : REAL;
		maxPeakCurrent : REAL;
		actCurrent : REAL;
		actVoltage : REAL;
		readPercentFromAccelerometer : BOOL := FALSE;
	END_STRUCT;
END_TYPE
```
